LIN {X 0,Y 576.248,Z 853.833,A -85,B 0,C 180,E1 -7834.379,E2 -7834.379} C_VEL
LIN {X 0,Y 576.344,Z 849.843,A -85,B 0,C 180,E1 -7836.475,E2 -7836.475} C_VEL
LIN {X 0,Y 576.515,Z 844.122,A -85,B 0,C 180,E1 -7838.578,E2 -7838.578} C_VEL
LIN {X 0,Y 576.818,Z 836.801,A -85,B 0,C 180,E1 -7840.618,E2 -7840.618} C_VEL
LIN {X 0,Y 577.289,Z 827.415,A -85,B 0,C 180,E1 -7842.707,E2 -7842.707} C_VEL
LIN {X 0,Y 577.934,Z 816.921,A -85,B 0,C 180,E1 -7844.631,E2 -7844.631} C_VEL
LIN {X 0,Y 578.818,Z 804.354,A -85,B 0,C 180,E1 -7846.561,E2 -7846.561} C_VEL
LIN {X 0,Y 579.816,Z 790.982,A -85,B 0,C 180,E1 -7848.292,E2 -7848.292} C_VEL
LIN {X 0,Y 580.962,Z 776.343,A -85,B 0,C 180,E1 -7849.924,E2 -7849.924} C_VEL
LIN {X 0,Y 582.298,Z 759.809,A -85,B 0,C 180,E1 -7851.507,E2 -7851.507} C_VEL
LIN {X 0,Y 583.711,Z 742.222,A -85,B 0,C 180,E1 -7852.946,E2 -7852.946} C_VEL
LIN {X 0,Y 585.156,Z 723.193,A -85,B 0,C 180,E1 -7854.265,E2 -7854.265} C_VEL
LIN {X 0,Y 586.509,Z 703.816,A -85,B 0,C 180,E1 -7855.389,E2 -7855.389} C_VEL
LIN {X 0,Y 587.764,Z 683.712,A -85,B 0,C 180,E1 -7856.36,E2 -7856.36} C_VEL
LIN {X 0,Y 588.932,Z 661.915,A -85,B 0,C 180,E1 -7857.211,E2 -7857.211} C_VEL
LIN {X 0,Y 589.873,Z 640.331,A -85,B 0,C 180,E1 -7857.867,E2 -7857.867} C_VEL
LIN {X 0,Y 590.601,Z 617.84,A -85,B 0,C 180,E1 -7858.365,E2 -7858.365} C_VEL
LIN {X 0,Y 594.551,Z 503.519,A -85,B 0,C 180,E1 -7860.286,E2 -7860.286} C_VEL
LIN {X 0,Y 597.181,Z 414.489,A -85,B 0,C 180,E1 -7861.618,E2 -7861.618} C_VEL
LIN {X 0,Y 598.837,Z 339.586,A -85,B 0,C 180,E1 -7862.637,E2 -7862.637} C_VEL
LIN {X 0,Y 599.448,Z 336.228,A -85,B 0,C 180,E1 -7862.787,E2 -7862.787} C_VEL
LIN {X 0,Y 599.375,Z 306.855,A -85,B 0,C 180,E1 -7864.729,E2 -7864.729} C_VEL
LIN {X 0,Y 600.383,Z 268.326,A -85,B 0,C 180,E1 -7867.502,E2 -7867.502} C_VEL
LIN {X 0,Y 591.929,Z 246.123,A -85,B 0,C 180,E1 -7869.848,E2 -7869.848} C_VEL
LIN {X 0,Y 584.236,Z 228.435,A -85,B 0,C 180,E1 -7871.74,E2 -7871.74} C_VEL
LIN {X 0,Y 578.995,Z 217.335,A -85,B 0,C 180,E1 -7872.927,E2 -7872.927} C_VEL
LIN {X 0,Y 577.607,Z 214.744,A -85,B 0,C 180,E1 -7873.215,E2 -7873.215} C_VEL
LIN {X 0,Y 577.299,Z 213.311,A -85,B 0,C 180,E1 -7873.366,E2 -7873.366} C_VEL
LIN {X 0,Y 577.308,Z 213.309,A -85,B 0,C 180,E1 -7876.696,E2 -7876.696} C_VEL
LIN {X 0,Y 577.314,Z 213.308,A -85,B 0,C 180,E1 -7879.954,E2 -7879.954} C_VEL
LIN {X 0,Y 577.298,Z 213.305,A -85,B 0,C 180,E1 -7883.182,E2 -7883.182} C_VEL
LIN {X 0,Y 577.315,Z 213.304,A -85,B 0,C 180,E1 -7886.461,E2 -7886.461} C_VEL
LIN {X 0,Y 577.32,Z 213.314,A -85,B 0,C 180,E1 -7889.85,E2 -7889.85} C_VEL
LIN {X 0,Y 577.304,Z 213.311,A -85,B 0,C 180,E1 -7893.124,E2 -7893.124} C_VEL
LIN {X 0,Y 577.307,Z 213.291,A -85,B 0,C 180,E1 -7896.416,E2 -7896.416} C_VEL
LIN {X 0,Y 577.316,Z 213.314,A -85,B 0,C 180,E1 -7899.733,E2 -7899.733} C_VEL
LIN {X 0,Y 577.309,Z 213.299,A -85,B 0,C 180,E1 -7903.084,E2 -7903.084} C_VEL
LIN {X 0,Y 577.3,Z 213.303,A -85,B 0,C 180,E1 -7906.326,E2 -7906.326} C_VEL
LIN {X 0,Y 577.315,Z 213.307,A -85,B 0,C 180,E1 -7909.659,E2 -7909.659} C_VEL
LIN {X 0,Y 577.319,Z 213.3,A -85,B 0,C 180,E1 -7913.036,E2 -7913.036} C_VEL
LIN {X 0,Y 577.297,Z 213.318,A -85,B 0,C 180,E1 -7916.326,E2 -7916.326} C_VEL
LIN {X 0,Y 577.313,Z 213.295,A -85,B 0,C 180,E1 -7919.603,E2 -7919.603} C_VEL
LIN {X 0,Y 577.307,Z 213.312,A -85,B 0,C 180,E1 -7922.879,E2 -7922.879} C_VEL
LIN {X 0,Y 577.294,Z 213.294,A -85,B 0,C 180,E1 -7926.182,E2 -7926.182} C_VEL
LIN {X 0,Y 577.317,Z 213.31,A -85,B 0,C 180,E1 -7929.47,E2 -7929.47} C_VEL
LIN {X 0,Y 577.291,Z 213.316,A -85,B 0,C 180,E1 -7932.707,E2 -7932.707} C_VEL
LIN {X 0,Y 577.307,Z 213.316,A -85,B 0,C 180,E1 -7936.001,E2 -7936.001} C_VEL
LIN {X 0,Y 577.319,Z 213.312,A -85,B 0,C 180,E1 -7939.318,E2 -7939.318} C_VEL
LIN {X 0,Y 577.283,Z 213.322,A -85,B 0,C 180,E1 -7942.506,E2 -7942.506} C_VEL
LIN {X 0,Y 577.32,Z 213.321,A -85,B 0,C 180,E1 -7945.768,E2 -7945.768} C_VEL
LIN {X 0,Y 577.294,Z 213.316,A -85,B 0,C 180,E1 -7949.011,E2 -7949.011} C_VEL
LIN {X 0,Y 577.282,Z 213.322,A -85,B 0,C 180,E1 -7952.358,E2 -7952.358} C_VEL
LIN {X 0,Y 577.322,Z 213.313,A -85,B 0,C 180,E1 -7955.587,E2 -7955.587} C_VEL
LIN {X 0,Y 577.271,Z 213.322,A -85,B 0,C 180,E1 -7958.79,E2 -7958.79} C_VEL
LIN {X 0,Y 577.318,Z 213.515,A -85,B 0,C 180,E1 -7959.175,E2 -7959.175} C_VEL
LIN {X 0,Y 578.825,Z 217.068,A -85,B 0,C 180,E1 -7959.601,E2 -7959.601} C_VEL
LIN {X 0,Y 588.305,Z 235.653,A -85,B 0,C 180,E1 -7961.909,E2 -7961.909} C_VEL
LIN {X 0,Y 600.676,Z 260.638,A -85,B 0,C 180,E1 -7964.76,E2 -7964.76} C_VEL
LIN {X 0,Y 607.806,Z 275.644,A -85,B 0,C 180,E1 -7966.338,E2 -7966.338} C_VEL
LIN {X 0,Y 605.103,Z 308.798,A -85,B 0,C 180,E1 -7968.172,E2 -7968.172} C_VEL
LIN {X 0,Y 607.829,Z 331.377,A -85,B 0,C 180,E1 -7968.729,E2 -7968.729} C_VEL
LIN {X 0,Y 602.232,Z 577.23,A -85,B 0,C 180,E1 -7972.119,E2 -7972.119} C_VEL
LIN {X 0,Y 599.928,Z 692.589,A -85,B 0,C 180,E1 -7973.674,E2 -7973.674} C_VEL
LIN {X 0,Y 598.876,Z 717.126,A -85,B 0,C 180,E1 -7974.167,E2 -7974.167} C_VEL
LIN {X 0,Y 597.663,Z 738.821,A -85,B 0,C 180,E1 -7974.744,E2 -7974.744} C_VEL
LIN {X 0,Y 596.011,Z 763.246,A -85,B 0,C 180,E1 -7975.572,E2 -7975.572} C_VEL
LIN {X 0,Y 594.427,Z 783.289,A -85,B 0,C 180,E1 -7976.399,E2 -7976.399} C_VEL
LIN {X 0,Y 592.413,Z 806.84,A -85,B 0,C 180,E1 -7977.556,E2 -7977.556} C_VEL
LIN {X 0,Y 590.599,Z 826.305,A -85,B 0,C 180,E1 -7978.684,E2 -7978.684} C_VEL
LIN {X 0,Y 588.459,Z 848.134,A -85,B 0,C 180,E1 -7980.142,E2 -7980.142} C_VEL
LIN {X 0,Y 586.519,Z 867.008,A -85,B 0,C 180,E1 -7981.603,E2 -7981.603} C_VEL
LIN {X 0,Y 584.495,Z 887.006,A -85,B 0,C 180,E1 -7983.372,E2 -7983.372} C_VEL
LIN {X 0,Y 582.762,Z 903.916,A -85,B 0,C 180,E1 -7985.088,E2 -7985.088} C_VEL
LIN {X 0,Y 581.074,Z 921.418,A -85,B 0,C 180,E1 -7987.114,E2 -7987.114} C_VEL
LIN {X 0,Y 579.75,Z 935.465,A -85,B 0,C 180,E1 -7988.977,E2 -7988.977} C_VEL
LIN {X 0,Y 578.56,Z 949.769,A -85,B 0,C 180,E1 -7991.145,E2 -7991.145} C_VEL
LIN {X 0,Y 577.681,Z 961.419,A -85,B 0,C 180,E1 -7993.199,E2 -7993.199} C_VEL
LIN {X 0,Y 576.975,Z 972.466,A -85,B 0,C 180,E1 -7995.447,E2 -7995.447} C_VEL
LIN {X 0,Y 576.545,Z 980.188,A -85,B 0,C 180,E1 -7997.378,E2 -7997.378} C_VEL
LIN {X 0,Y 576.225,Z 987.119,A -85,B 0,C 180,E1 -7999.502,E2 -7999.502} C_VEL
LIN {X 0,Y 576.012,Z 993.449,A -85,B 0,C 180,E1 -8001.917,E2 -8001.917} C_VEL
LIN {X 0,Y 575.941,Z 997.697,A -85,B 0,C 180,E1 -8004.148,E2 -8004.148} C_VEL
LIN {X 0,Y 575.915,Z 1000.576,A -85,B 0,C 180,E1 -8006.317,E2 -8006.317} C_VEL
LIN {X 0,Y 575.907,Z 1002.235,A -85,B 0,C 180,E1 -8008.806,E2 -8008.806} C_VEL
LIN {X 0,Y 575.888,Z 1002.325,A -85,B 0,C 180,E1 -8010.796,E2 -8010.796} C_VEL
LIN {X 0,Y 575.886,Z 1001.289,A -85,B 0,C 180,E1 -8012.886,E2 -8012.886} C_VEL
LIN {X 0,Y 575.909,Z 998.45,A -85,B 0,C 180,E1 -8015.38,E2 -8015.38} C_VEL
LIN {X 0,Y 575.969,Z 994.688,A -85,B 0,C 180,E1 -8017.481,E2 -8017.481} C_VEL
LIN {X 0,Y 576.141,Z 989.457,A -85,B 0,C 180,E1 -8019.692,E2 -8019.692} C_VEL
LIN {X 0,Y 576.451,Z 981.951,A -85,B 0,C 180,E1 -8022.116,E2 -8022.116} C_VEL
LIN {X 0,Y 576.79,Z 975.298,A -85,B 0,C 180,E1 -8023.883,E2 -8023.883} C_VEL
LIN {X 0,Y 577.322,Z 966.57,A -85,B 0,C 180,E1 -8025.778,E2 -8025.778} C_VEL
LIN {X 0,Y 578.171,Z 954.305,A -85,B 0,C 180,E1 -8028.033,E2 -8028.033} C_VEL
LIN {X 0,Y 579.14,Z 941.931,A -85,B 0,C 180,E1 -8029.99,E2 -8029.99} C_VEL
LIN {X 0,Y 580.46,Z 926.019,A -85,B 0,C 180,E1 -8032.163,E2 -8032.163} C_VEL
LIN {X 0,Y 581.785,Z 911.136,A -85,B 0,C 180,E1 -8033.929,E2 -8033.929} C_VEL
LIN {X 0,Y 583.484,Z 892.287,A -85,B 0,C 180,E1 -8035.885,E2 -8035.885} C_VEL
LIN {X 0,Y 585.062,Z 875.137,A -85,B 0,C 180,E1 -8037.432,E2 -8037.432} C_VEL
LIN {X 0,Y 586.934,Z 854.247,A -85,B 0,C 180,E1 -8039.08,E2 -8039.08} C_VEL
LIN {X 0,Y 588.596,Z 834.717,A -85,B 0,C 180,E1 -8040.413,E2 -8040.413} C_VEL
LIN {X 0,Y 590.519,Z 811.335,A -85,B 0,C 180,E1 -8041.787,E2 -8041.787} C_VEL
LIN {X 0,Y 592.038,Z 790.551,A -85,B 0,C 180,E1 -8042.829,E2 -8042.829} C_VEL
LIN {X 0,Y 593.635,Z 766.597,A -85,B 0,C 180,E1 -8043.832,E2 -8043.832} C_VEL
LIN {X 0,Y 594.899,Z 744.933,A -85,B 0,C 180,E1 -8044.58,E2 -8044.58} C_VEL
LIN {X 0,Y 596.12,Z 719.728,A -85,B 0,C 180,E1 -8045.261,E2 -8045.261} C_VEL
LIN {X 0,Y 596.892,Z 698.83,A -85,B 0,C 180,E1 -8045.688,E2 -8045.688} C_VEL
LIN {X 0,Y 597.508,Z 665.557,A -85,B 0,C 180,E1 -8046.153,E2 -8046.153} C_VEL
LIN {X 0,Y 599.383,Z 523.368,A -85,B 0,C 180,E1 -8047.959,E2 -8047.959} C_VEL
LIN {X 0,Y 602.037,Z 398.059,A -85,B 0,C 180,E1 -8049.719,E2 -8049.719} C_VEL
LIN {X 0,Y 603.978,Z 328.15,A -85,B 0,C 180,E1 -8050.796,E2 -8050.796} C_VEL
LIN {X 0,Y 603.753,Z 324.587,A -85,B 0,C 180,E1 -8050.92,E2 -8050.92} C_VEL
LIN {X 0,Y 608.265,Z 300.685,A -85,B 0,C 180,E1 -8052.571,E2 -8052.571} C_VEL
LIN {X 0,Y 613.531,Z 280.646,A -85,B 0,C 180,E1 -8054.099,E2 -8054.099} C_VEL
LIN {X 0,Y 612.091,Z 275.219,A -85,B 0,C 180,E1 -8055.284,E2 -8055.284} C_VEL
LIN {X 0,Y 611.11,Z 271.585,A -85,B 0,C 180,E1 -8056.462,E2 -8056.462} C_VEL
LIN {X 0,Y 610.691,Z 269.324,A -85,B 0,C 180,E1 -8057.877,E2 -8057.877} C_VEL
LIN {X 0,Y 610.625,Z 269.272,A -85,B 0,C 180,E1 -8058.457,E2 -8058.457} C_VEL
LIN {X 0,Y 610.726,Z 271.372,A -85,B 0,C 180,E1 -8059.952,E2 -8059.952} C_VEL
LIN {X 0,Y 611.329,Z 275.332,A -85,B 0,C 180,E1 -8061.212,E2 -8061.212} C_VEL
LIN {X 0,Y 611.672,Z 278.803,A -85,B 0,C 180,E1 -8061.955,E2 -8061.955} C_VEL
LIN {X 0,Y 605.574,Z 300.252,A -85,B 0,C 180,E1 -8063.881,E2 -8063.881} C_VEL
LIN {X 0,Y 599.965,Z 327.92,A -85,B 0,C 180,E1 -8066.176,E2 -8066.176} C_VEL
LIN {X 0,Y 595.013,Z 362.924,A -85,B 0,C 180,E1 -8068.886,E2 -8068.886} C_VEL
LIN {X 0,Y 590.47,Z 407.602,A -85,B 0,C 180,E1 -8072.122,E2 -8072.122} C_VEL
LIN {X 0,Y 589.4,Z 422.994,A -85,B 0,C 180,E1 -8073.168,E2 -8073.168} C_VEL
LIN {X 0,Y 592.686,Z 455.008,A -85,B 0,C 180,E1 -8074.339,E2 -8074.339} C_VEL
LIN {X 0,Y 595.543,Z 491.146,A -85,B 0,C 180,E1 -8075.476,E2 -8075.476} C_VEL
LIN {X 0,Y 594.867,Z 505.645,A -85,B 0,C 180,E1 -8075.78,E2 -8075.78} C_VEL
LIN {X 0,Y 589.455,Z 607.464,A -85,B 0,C 180,E1 -8077.73,E2 -8077.73} C_VEL
LIN {X 0,Y 586.293,Z 687.572,A -85,B 0,C 180,E1 -8079.223,E2 -8079.223} C_VEL
LIN {X 0,Y 585.33,Z 709.905,A -85,B 0,C 180,E1 -8079.833,E2 -8079.833} C_VEL
LIN {X 0,Y 584.359,Z 731.272,A -85,B 0,C 180,E1 -8080.613,E2 -8080.613} C_VEL
LIN {X 0,Y 583.386,Z 750.706,A -85,B 0,C 180,E1 -8081.514,E2 -8081.514} C_VEL
LIN {X 0,Y 582.433,Z 769.003,A -85,B 0,C 180,E1 -8082.568,E2 -8082.568} C_VEL
LIN {X 0,Y 581.473,Z 786.178,A -85,B 0,C 180,E1 -8083.774,E2 -8083.774} C_VEL
LIN {X 0,Y 580.594,Z 801.262,A -85,B 0,C 180,E1 -8085.049,E2 -8085.049} C_VEL
LIN {X 0,Y 579.773,Z 814.876,A -85,B 0,C 180,E1 -8086.435,E2 -8086.435} C_VEL
LIN {X 0,Y 579.038,Z 827.147,A -85,B 0,C 180,E1 -8087.939,E2 -8087.939} C_VEL
LIN {X 0,Y 578.439,Z 837.273,A -85,B 0,C 180,E1 -8089.442,E2 -8089.442} C_VEL
LIN {X 0,Y 577.896,Z 846.496,A -85,B 0,C 180,E1 -8091.142,E2 -8091.142} C_VEL
LIN {X 0,Y 577.499,Z 853.707,A -85,B 0,C 180,E1 -8092.839,E2 -8092.839} C_VEL
LIN {X 0,Y 577.21,Z 859.389,A -85,B 0,C 180,E1 -8094.632,E2 -8094.632} C_VEL
LIN {X 0,Y 576.993,Z 863.232,A -85,B 0,C 180,E1 -8096.423,E2 -8096.423} C_VEL
LIN {X 0,Y 576.852,Z 865.342,A -85,B 0,C 180,E1 -8098.212,E2 -8098.212} C_VEL
LIN {X 0,Y 576.771,Z 865.736,A -85,B 0,C 180,E1 -8100.099,E2 -8100.099} C_VEL
LIN {X 0,Y 576.736,Z 864.293,A -85,B 0,C 180,E1 -8101.987,E2 -8101.987} C_VEL
LIN {X 0,Y 576.764,Z 861.014,A -85,B 0,C 180,E1 -8103.877,E2 -8103.877} C_VEL
LIN {X 0,Y 576.874,Z 856.161,A -85,B 0,C 180,E1 -8105.67,E2 -8105.67} C_VEL
LIN {X 0,Y 577.061,Z 849.471,A -85,B 0,C 180,E1 -8107.467,E2 -8107.467} C_VEL
LIN {X 0,Y 577.367,Z 841.126,A -85,B 0,C 180,E1 -8109.201,E2 -8109.201} C_VEL
LIN {X 0,Y 577.814,Z 831.101,A -85,B 0,C 180,E1 -8110.872,E2 -8110.872} C_VEL
LIN {X 0,Y 578.397,Z 819.329,A -85,B 0,C 180,E1 -8112.48,E2 -8112.48} C_VEL
LIN {X 0,Y 579.11,Z 805.98,A -85,B 0,C 180,E1 -8113.988,E2 -8113.988} C_VEL
LIN {X 0,Y 579.937,Z 790.987,A -85,B 0,C 180,E1 -8115.398,E2 -8115.398} C_VEL
LIN {X 0,Y 580.827,Z 774.875,A -85,B 0,C 180,E1 -8116.656,E2 -8116.656} C_VEL
LIN {X 0,Y 581.733,Z 757.436,A -85,B 0,C 180,E1 -8117.782,E2 -8117.782} C_VEL
LIN {X 0,Y 582.635,Z 739.626,A -85,B 0,C 180,E1 -8118.719,E2 -8118.719} C_VEL
LIN {X 0,Y 583.514,Z 720.275,A -85,B 0,C 180,E1 -8119.531,E2 -8119.531} C_VEL
LIN {X 0,Y 584.279,Z 700.12,A -85,B 0,C 180,E1 -8120.172,E2 -8120.172} C_VEL
LIN {X 0,Y 584.919,Z 679.428,A -85,B 0,C 180,E1 -8120.63,E2 -8120.63} C_VEL
LIN {X 0,Y 588.981,Z 489.215,A -85,B 0,C 180,E1 -8123.466,E2 -8123.466} C_VEL
LIN {X 0,Y 585.221,Z 455.543,A -85,B 0,C 180,E1 -8124.209,E2 -8124.209} C_VEL
LIN {X 0,Y 587.587,Z 405.605,A -85,B 0,C 180,E1 -8127.406,E2 -8127.406} C_VEL
LIN {X 0,Y 590.441,Z 352.546,A -85,B 0,C 180,E1 -8130.842,E2 -8130.842} C_VEL
LIN {X 0,Y 593.46,Z 300.77,A -85,B 0,C 180,E1 -8134.246,E2 -8134.246} C_VEL
LIN {X 0,Y 595.914,Z 261.134,A -85,B 0,C 180,E1 -8136.892,E2 -8136.892} C_VEL
LIN {X 0,Y 591.877,Z 250.242,A -85,B 0,C 180,E1 -8137.944,E2 -8137.944} C_VEL
LIN {X 0,Y 589.101,Z 245.546,A -85,B 0,C 180,E1 -8138.478,E2 -8138.478} C_VEL
LIN {X 0,Y 577.793,Z 233.961,A -85,B 0,C 180,E1 -8140.148,E2 -8140.148} C_VEL
LIN {X 0,Y 576.198,Z 231.311,A -85,B 0,C 180,E1 -8140.468,E2 -8140.468} C_VEL
LIN {X 0,Y 569.344,Z 214.421,A -85,B 0,C 180,E1 -8142.302,E2 -8142.302} C_VEL
LIN {X 0,Y 569.381,Z 214.302,A -85,B 0,C 180,E1 -8145.518,E2 -8145.518} C_VEL
LIN {X 0,Y 569.39,Z 214.435,A -85,B 0,C 180,E1 -8146.119,E2 -8146.119} C_VEL
LIN {X 0,Y 570.341,Z 217.235,A -85,B 0,C 180,E1 -8146.39,E2 -8146.39} C_VEL
LIN {X 0,Y 571.71,Z 219.791,A -85,B 0,C 180,E1 -8146.683,E2 -8146.683} C_VEL
LIN {X 0,Y 578.876,Z 234.711,A -85,B 0,C 180,E1 -8148.317,E2 -8148.317} C_VEL
LIN {X 0,Y 586.838,Z 253.704,A -85,B 0,C 180,E1 -8150.367,E2 -8150.367} C_VEL
LIN {X 0,Y 593.746,Z 272.147,A -85,B 0,C 180,E1 -8152.326,E2 -8152.326} C_VEL
LIN {X 0,Y 592.76,Z 314.667,A -85,B 0,C 180,E1 -8155.357,E2 -8155.357} C_VEL
LIN {X 0,Y 592.824,Z 338.961,A -85,B 0,C 180,E1 -8156.932,E2 -8156.932} C_VEL
LIN {X 0,Y 591.933,Z 343.747,A -85,B 0,C 180,E1 -8157.101,E2 -8157.101} C_VEL
LIN {X 0,Y 589.728,Z 439.794,A -85,B 0,C 180,E1 -8158.419,E2 -8158.419} C_VEL
LIN {X 0,Y 586.74,Z 530.066,A -85,B 0,C 180,E1 -8159.837,E2 -8159.837} C_VEL
LIN {X 0,Y 583.259,Z 625.148,A -85,B 0,C 180,E1 -8161.508,E2 -8161.508} C_VEL
LIN {X 0,Y 582.489,Z 647.168,A -85,B 0,C 180,E1 -8162.048,E2 -8162.048} C_VEL
LIN {X 0,Y 581.453,Z 668.771,A -85,B 0,C 180,E1 -8162.755,E2 -8162.755} C_VEL
LIN {X 0,Y 580.207,Z 690.159,A -85,B 0,C 180,E1 -8163.655,E2 -8163.655} C_VEL
LIN {X 0,Y 578.823,Z 710.131,A -85,B 0,C 180,E1 -8164.688,E2 -8164.688} C_VEL
LIN {X 0,Y 577.378,Z 729.317,A -85,B 0,C 180,E1 -8165.877,E2 -8165.877} C_VEL
LIN {X 0,Y 575.82,Z 748.322,A -85,B 0,C 180,E1 -8167.272,E2 -8167.272} C_VEL
LIN {X 0,Y 574.417,Z 765.121,A -85,B 0,C 180,E1 -8168.719,E2 -8168.719} C_VEL
LIN {X 0,Y 573.057,Z 781.033,A -85,B 0,C 180,E1 -8170.321,E2 -8170.321} C_VEL
LIN {X 0,Y 571.809,Z 795.88,A -85,B 0,C 180,E1 -8172.076,E2 -8172.076} C_VEL
LIN {X 0,Y 570.757,Z 809.256,A -85,B 0,C 180,E1 -8173.931,E2 -8173.931} C_VEL
LIN {X 0,Y 569.863,Z 821.736,A -85,B 0,C 180,E1 -8175.987,E2 -8175.987} C_VEL
LIN {X 0,Y 569.248,Z 831.607,A -85,B 0,C 180,E1 -8177.935,E2 -8177.935} C_VEL
LIN {X 0,Y 568.806,Z 840.094,A -85,B 0,C 180,E1 -8179.978,E2 -8179.978} C_VEL
LIN {X 0,Y 568.521,Z 846.753,A -85,B 0,C 180,E1 -8182.013,E2 -8182.013} C_VEL
LIN {X 0,Y 568.361,Z 852.257,A -85,B 0,C 180,E1 -8184.245,E2 -8184.245} C_VEL
LIN {X 0,Y 568.297,Z 855.835,A -85,B 0,C 180,E1 -8186.368,E2 -8186.368} C_VEL
LIN {X 0,Y 568.26,Z 857.744,A -85,B 0,C 180,E1 -8188.488,E2 -8188.488} C_VEL
LIN {X 0,Y 568.247,Z 858.093,A -85,B 0,C 180,E1 -8190.605,E2 -8190.605} C_VEL
LIN {X 0,Y 568.274,Z 856.938,A -85,B 0,C 180,E1 -8192.723,E2 -8192.723} C_VEL
LIN {X 0,Y 568.33,Z 854.144,A -85,B 0,C 180,E1 -8194.844,E2 -8194.844} C_VEL
LIN {X 0,Y 568.421,Z 849.713,A -85,B 0,C 180,E1 -8196.971,E2 -8196.971} C_VEL
LIN {X 0,Y 568.641,Z 843.588,A -85,B 0,C 180,E1 -8199.106,E2 -8199.106} C_VEL
LIN {X 0,Y 569.027,Z 836.048,A -85,B 0,C 180,E1 -8201.145,E2 -8201.145} C_VEL
LIN {X 0,Y 569.547,Z 826.578,A -85,B 0,C 180,E1 -8203.193,E2 -8203.193} C_VEL
LIN {X 0,Y 570.279,Z 815.707,A -85,B 0,C 180,E1 -8205.144,E2 -8205.144} C_VEL
LIN {X 0,Y 571.203,Z 803.495,A -85,B 0,C 180,E1 -8206.998,E2 -8206.998} C_VEL
LIN {X 0,Y 572.319,Z 789.976,A -85,B 0,C 180,E1 -8208.751,E2 -8208.751} C_VEL
LIN {X 0,Y 573.661,Z 774.003,A -85,B 0,C 180,E1 -8210.508,E2 -8210.508} C_VEL
LIN {X 0,Y 575.071,Z 757.356,A -85,B 0,C 180,E1 -8212.067,E2 -8212.067} C_VEL
LIN {X 0,Y 576.568,Z 739.348,A -85,B 0,C 180,E1 -8213.507,E2 -8213.507} C_VEL
LIN {X 0,Y 578.148,Z 719.445,A -85,B 0,C 180,E1 -8214.851,E2 -8214.851} C_VEL
LIN {X 0,Y 579.515,Z 700.296,A -85,B 0,C 180,E1 -8215.937,E2 -8215.937} C_VEL
LIN {X 0,Y 580.878,Z 679.328,A -85,B 0,C 180,E1 -8216.918,E2 -8216.918} C_VEL
LIN {X 0,Y 581.989,Z 658.553,A -85,B 0,C 180,E1 -8217.693,E2 -8217.693} C_VEL
LIN {X 0,Y 582.878,Z 636.878,A -85,B 0,C 180,E1 -8218.318,E2 -8218.318} C_VEL
LIN {X 0,Y 583.753,Z 609.709,A -85,B 0,C 180,E1 -8218.876,E2 -8218.876} C_VEL
LIN {X 0,Y 587.697,Z 503.594,A -85,B 0,C 180,E1 -8220.688,E2 -8220.688} C_VEL
LIN {X 0,Y 590.36,Z 417.842,A -85,B 0,C 180,E1 -8221.989,E2 -8221.989} C_VEL
LIN {X 0,Y 591.983,Z 342.833,A -85,B 0,C 180,E1 -8223.005,E2 -8223.005} C_VEL
LIN {X 0,Y 592.926,Z 337.654,A -85,B 0,C 180,E1 -8223.235,E2 -8223.235} C_VEL
LIN {X 0,Y 592.875,Z 307.651,A -85,B 0,C 180,E1 -8225.225,E2 -8225.225} C_VEL
LIN {X 0,Y 593.748,Z 271.834,A -85,B 0,C 180,E1 -8227.806,E2 -8227.806} C_VEL
LIN {X 0,Y 585.364,Z 249.888,A -85,B 0,C 180,E1 -8230.146,E2 -8230.146} C_VEL
LIN {X 0,Y 578.158,Z 233.181,A -85,B 0,C 180,E1 -8231.956,E2 -8231.956} C_VEL
LIN {X 0,Y 571.21,Z 218.485,A -85,B 0,C 180,E1 -8233.556,E2 -8233.556} C_VEL
LIN {X 0,Y 569.605,Z 215.436,A -85,B 0,C 180,E1 -8233.899,E2 -8233.899} C_VEL
LIN {X 0,Y 569.377,Z 214.299,A -85,B 0,C 180,E1 -8234.026,E2 -8234.026} C_VEL
LIN {X 0,Y 569.36,Z 214.306,A -85,B 0,C 180,E1 -8237.322,E2 -8237.322} C_VEL
LIN {X 0,Y 569.378,Z 214.305,A -85,B 0,C 180,E1 -8240.657,E2 -8240.657} C_VEL
LIN {X 0,Y 569.374,Z 214.297,A -85,B 0,C 180,E1 -8243.963,E2 -8243.963} C_VEL
LIN {X 0,Y 569.361,Z 214.289,A -85,B 0,C 180,E1 -8247.267,E2 -8247.267} C_VEL
LIN {X 0,Y 569.38,Z 214.295,A -85,B 0,C 180,E1 -8250.578,E2 -8250.578} C_VEL
LIN {X 0,Y 569.374,Z 214.308,A -85,B 0,C 180,E1 -8253.958,E2 -8253.958} C_VEL
LIN {X 0,Y 569.365,Z 214.284,A -85,B 0,C 180,E1 -8257.272,E2 -8257.272} C_VEL
LIN {X 0,Y 569.371,Z 214.293,A -85,B 0,C 180,E1 -8260.569,E2 -8260.569} C_VEL
LIN {X 0,Y 569.372,Z 214.303,A -85,B 0,C 180,E1 -8263.995,E2 -8263.995} C_VEL
LIN {X 0,Y 569.369,Z 214.281,A -85,B 0,C 180,E1 -8267.216,E2 -8267.216} C_VEL
LIN {X 0,Y 569.363,Z 214.305,A -85,B 0,C 180,E1 -8270.498,E2 -8270.498} C_VEL
LIN {X 0,Y 569.374,Z 214.277,A -85,B 0,C 180,E1 -8273.85,E2 -8273.85} C_VEL
LIN {X 0,Y 569.376,Z 214.304,A -85,B 0,C 180,E1 -8277.182,E2 -8277.182} C_VEL
LIN {X 0,Y 569.352,Z 214.275,A -85,B 0,C 180,E1 -8280.402,E2 -8280.402} C_VEL
LIN {X 0,Y 569.376,Z 214.308,A -85,B 0,C 180,E1 -8283.725,E2 -8283.725} C_VEL
LIN {X 0,Y 569.38,Z 214.272,A -85,B 0,C 180,E1 -8287.061,E2 -8287.061} C_VEL
LIN {X 0,Y 569.35,Z 214.308,A -85,B 0,C 180,E1 -8290.422,E2 -8290.422} C_VEL
LIN {X 0,Y 569.382,Z 214.308,A -85,B 0,C 180,E1 -8293.714,E2 -8293.714} C_VEL
LIN {X 0,Y 569.361,Z 214.306,A -85,B 0,C 180,E1 -8296.949,E2 -8296.949} C_VEL
LIN {X 0,Y 569.348,Z 214.308,A -85,B 0,C 180,E1 -8300.349,E2 -8300.349} C_VEL
LIN {X 0,Y 569.383,Z 214.305,A -85,B 0,C 180,E1 -8303.603,E2 -8303.603} C_VEL
LIN {X 0,Y 569.346,Z 214.301,A -85,B 0,C 180,E1 -8306.855,E2 -8306.855} C_VEL
LIN {X 0,Y 569.353,Z 214.312,A -85,B 0,C 180,E1 -8310.226,E2 -8310.226} C_VEL
LIN {X 0,Y 569.381,Z 214.303,A -85,B 0,C 180,E1 -8313.473,E2 -8313.473} C_VEL
LIN {X 0,Y 569.334,Z 214.309,A -85,B 0,C 180,E1 -8316.664,E2 -8316.664} C_VEL
LIN {X 0,Y 569.358,Z 214.444,A -85,B 0,C 180,E1 -8318.406,E2 -8318.406} C_VEL
LIN {X 0,Y 570.387,Z 217.397,A -85,B 0,C 180,E1 -8318.743,E2 -8318.743} C_VEL
LIN {X 0,Y 571.764,Z 219.658,A -85,B 0,C 180,E1 -8319.063,E2 -8319.063} C_VEL
LIN {X 0,Y 581.042,Z 238.068,A -85,B 0,C 180,E1 -8321.384,E2 -8321.384} C_VEL
LIN {X 0,Y 592.456,Z 260.848,A -85,B 0,C 180,E1 -8324.054,E2 -8324.054} C_VEL
LIN {X 0,Y 601.171,Z 279.402,A -85,B 0,C 180,E1 -8326.036,E2 -8326.036} C_VEL
LIN {X 0,Y 598.614,Z 309.394,A -85,B 0,C 180,E1 -8327.71,E2 -8327.71} C_VEL
LIN {X 0,Y 601.382,Z 332.717,A -85,B 0,C 180,E1 -8328.291,E2 -8328.291} C_VEL
LIN {X 0,Y 595.541,Z 572.332,A -85,B 0,C 180,E1 -8331.646,E2 -8331.646} C_VEL
LIN {X 0,Y 592.986,Z 692.835,A -85,B 0,C 180,E1 -8333.293,E2 -8333.293} C_VEL
LIN {X 0,Y 591.882,Z 717.267,A -85,B 0,C 180,E1 -8333.79,E2 -8333.79} C_VEL
LIN {X 0,Y 590.638,Z 738.58,A -85,B 0,C 180,E1 -8334.363,E2 -8334.363} C_VEL
LIN {X 0,Y 588.881,Z 763.35,A -85,B 0,C 180,E1 -8335.214,E2 -8335.214} C_VEL
LIN {X 0,Y 587.231,Z 783.315,A -85,B 0,C 180,E1 -8336.048,E2 -8336.048} C_VEL
LIN {X 0,Y 585.054,Z 807.455,A -85,B 0,C 180,E1 -8337.254,E2 -8337.254} C_VEL
LIN {X 0,Y 583.145,Z 827.122,A -85,B 0,C 180,E1 -8338.411,E2 -8338.411} C_VEL
LIN {X 0,Y 580.833,Z 849.426,A -85,B 0,C 180,E1 -8339.937,E2 -8339.937} C_VEL
LIN {X 0,Y 578.942,Z 867.051,A -85,B 0,C 180,E1 -8341.327,E2 -8341.327} C_VEL
LIN {X 0,Y 576.775,Z 887.323,A -85,B 0,C 180,E1 -8343.154,E2 -8343.154} C_VEL
LIN {X 0,Y 575.028,Z 903.654,A -85,B 0,C 180,E1 -8344.84,E2 -8344.84} C_VEL
LIN {X 0,Y 573.254,Z 921.098,A -85,B 0,C 180,E1 -8346.893,E2 -8346.893} C_VEL
LIN {X 0,Y 571.882,Z 935.11,A -85,B 0,C 180,E1 -8348.782,E2 -8348.782} C_VEL
LIN {X 0,Y 570.586,Z 949.964,A -85,B 0,C 180,E1 -8351.083,E2 -8351.083} C_VEL
LIN {X 0,Y 569.728,Z 960.976,A -85,B 0,C 180,E1 -8353.062,E2 -8353.062} C_VEL
LIN {X 0,Y 568.973,Z 972.391,A -85,B 0,C 180,E1 -8355.445,E2 -8355.445} C_VEL
LIN {X 0,Y 568.499,Z 980.992,A -85,B 0,C 180,E1 -8357.609,E2 -8357.609} C_VEL
LIN {X 0,Y 568.169,Z 988.802,A -85,B 0,C 180,E1 -8359.967,E2 -8359.967} C_VEL
LIN {X 0,Y 567.986,Z 994.275,A -85,B 0,C 180,E1 -8362.21,E2 -8362.21} C_VEL
LIN {X 0,Y 567.934,Z 997.972,A -85,B 0,C 180,E1 -8364.241,E2 -8364.241} C_VEL
LIN {X 0,Y 567.903,Z 1001.015,A -85,B 0,C 180,E1 -8366.669,E2 -8366.669} C_VEL
LIN {X 0,Y 567.898,Z 1002.28,A -85,B 0,C 180,E1 -8368.991,E2 -8368.991} C_VEL
LIN {X 0,Y 567.898,Z 1002.28,A -85,B 0,C 180,E1 -8371.009,E2 -8371.009} C_VEL
LIN {X 0,Y 567.906,Z 1000.915,A -85,B 0,C 180,E1 -8373.432,E2 -8373.432} C_VEL
LIN {X 0,Y 567.934,Z 997.971,A -85,B 0,C 180,E1 -8375.76,E2 -8375.76} C_VEL
LIN {X 0,Y 567.993,Z 994.069,A -85,B 0,C 180,E1 -8377.892,E2 -8377.892} C_VEL
LIN {X 0,Y 568.191,Z 988.158,A -85,B 0,C 180,E1 -8380.238,E2 -8380.238} C_VEL
LIN {X 0,Y 568.5,Z 980.91,A -85,B 0,C 180,E1 -8382.391,E2 -8382.391} C_VEL
LIN {X 0,Y 568.978,Z 972.186,A -85,B 0,C 180,E1 -8384.555,E2 -8384.555} C_VEL
LIN {X 0,Y 569.688,Z 961.092,A -85,B 0,C 180,E1 -8386.834,E2 -8386.834} C_VEL
LIN {X 0,Y 570.533,Z 949.674,A -85,B 0,C 180,E1 -8388.847,E2 -8388.847} C_VEL
LIN {X 0,Y 571.694,Z 935.436,A -85,B 0,C 180,E1 -8391.011,E2 -8391.011} C_VEL
LIN {X 0,Y 572.997,Z 921.077,A -85,B 0,C 180,E1 -8392.901,E2 -8392.901} C_VEL
LIN {X 0,Y 574.602,Z 903.659,A -85,B 0,C 180,E1 -8394.905,E2 -8394.905} C_VEL
LIN {X 0,Y 576.157,Z 887.303,A -85,B 0,C 180,E1 -8396.544,E2 -8396.544} C_VEL
LIN {X 0,Y 577.957,Z 868.083,A -85,B 0,C 180,E1 -8398.24,E2 -8398.24} C_VEL
LIN {X 0,Y 579.754,Z 848.643,A -85,B 0,C 180,E1 -8399.726,E2 -8399.726} C_VEL
LIN {X 0,Y 581.774,Z 826.231,A -85,B 0,C 180,E1 -8401.211,E2 -8401.211} C_VEL
LIN {X 0,Y 583.371,Z 806.617,A -85,B 0,C 180,E1 -8402.328,E2 -8402.328} C_VEL
LIN {X 0,Y 585.213,Z 782.574,A -85,B 0,C 180,E1 -8403.496,E2 -8403.496} C_VEL
LIN {X 0,Y 586.653,Z 761.498,A -85,B 0,C 180,E1 -8404.344,E2 -8404.344} C_VEL
LIN {X 0,Y 588.123,Z 736.576,A -85,B 0,C 180,E1 -8405.164,E2 -8405.164} C_VEL
LIN {X 0,Y 589.14,Z 714.548,A -85,B 0,C 180,E1 -8405.726,E2 -8405.726} C_VEL
LIN {X 0,Y 590.03,Z 688.498,A -85,B 0,C 180,E1 -8406.211,E2 -8406.211} C_VEL
LIN {X 0,Y 592.517,Z 526.417,A -85,B 0,C 180,E1 -8408.323,E2 -8408.323} C_VEL
LIN {X 0,Y 595.353,Z 407.844,A -85,B 0,C 180,E1 -8410.036,E2 -8410.036} C_VEL
LIN {X 0,Y 597.915,Z 329.601,A -85,B 0,C 180,E1 -8411.28,E2 -8411.28} C_VEL
LIN {X 0,Y 597.763,Z 327.352,A -85,B 0,C 180,E1 -8411.355,E2 -8411.355} C_VEL
LIN {X 0,Y 602.798,Z 303.687,A -85,B 0,C 180,E1 -8413.045,E2 -8413.045} C_VEL
LIN {X 0,Y 608.154,Z 285.464,A -85,B 0,C 180,E1 -8414.475,E2 -8414.475} C_VEL
LIN {X 0,Y 607.008,Z 280.361,A -85,B 0,C 180,E1 -8415.698,E2 -8415.698} C_VEL
LIN {X 0,Y 606.272,Z 277.736,A -85,B 0,C 180,E1 -8416.679,E2 -8416.679} C_VEL
LIN {X 0,Y 606.126,Z 275.632,A -85,B 0,C 180,E1 -8418.214,E2 -8418.214} C_VEL
LIN {X 0,Y 605.897,Z 277.499,A -85,B 0,C 180,E1 -8419.691,E2 -8419.691} C_VEL
LIN {X 0,Y 606.251,Z 280.584,A -85,B 0,C 180,E1 -8420.825,E2 -8420.825} C_VEL
LIN {X 0,Y 606.491,Z 283.655,A -85,B 0,C 180,E1 -8421.571,E2 -8421.571} C_VEL
LIN {X 0,Y 599.82,Z 304.959,A -85,B 0,C 180,E1 -8423.538,E2 -8423.538} C_VEL
LIN {X 0,Y 593.809,Z 331.937,A -85,B 0,C 180,E1 -8425.836,E2 -8425.836} C_VEL
LIN {X 0,Y 588.656,Z 364.932,A -85,B 0,C 180,E1 -8428.455,E2 -8428.455} C_VEL
LIN {X 0,Y 583.914,Z 406.935,A -85,B 0,C 180,E1 -8431.572,E2 -8431.572} C_VEL
LIN {X 0,Y 582.884,Z 419.506,A -85,B 0,C 180,E1 -8432.447,E2 -8432.447} C_VEL
LIN {X 0,Y 585.632,Z 446.596,A -85,B 0,C 180,E1 -8433.505,E2 -8433.505} C_VEL
LIN {X 0,Y 588.405,Z 481.333,A -85,B 0,C 180,E1 -8434.69,E2 -8434.69} C_VEL
LIN {X 0,Y 589.088,Z 495.815,A -85,B 0,C 180,E1 -8435.116,E2 -8435.116} C_VEL
LIN {X 0,Y 583.019,Z 598.12,A -85,B 0,C 180,E1 -8437.152,E2 -8437.152} C_VEL
LIN {X 0,Y 579.118,Z 687.482,A -85,B 0,C 180,E1 -8438.87,E2 -8438.87} C_VEL
LIN {X 0,Y 578.059,Z 710.48,A -85,B 0,C 180,E1 -8439.509,E2 -8439.509} C_VEL
LIN {X 0,Y 577.073,Z 730.613,A -85,B 0,C 180,E1 -8440.252,E2 -8440.252} C_VEL
LIN {X 0,Y 576.021,Z 750.164,A -85,B 0,C 180,E1 -8441.163,E2 -8441.163} C_VEL
LIN {X 0,Y 575.015,Z 768.532,A -85,B 0,C 180,E1 -8442.215,E2 -8442.215} C_VEL
LIN {X 0,Y 574.02,Z 785.524,A -85,B 0,C 180,E1 -8443.401,E2 -8443.401} C_VEL
LIN {X 0,Y 573.042,Z 801.208,A -85,B 0,C 180,E1 -8444.723,E2 -8444.723} C_VEL
LIN {X 0,Y 572.151,Z 815.237,A -85,B 0,C 180,E1 -8446.148,E2 -8446.148} C_VEL
LIN {X 0,Y 571.352,Z 827.64,A -85,B 0,C 180,E1 -8447.672,E2 -8447.672} C_VEL
LIN {X 0,Y 570.654,Z 838.462,A -85,B 0,C 180,E1 -8449.296,E2 -8449.296} C_VEL
LIN {X 0,Y 570.107,Z 847.239,A -85,B 0,C 180,E1 -8450.918,E2 -8450.918} C_VEL
LIN {X 0,Y 569.668,Z 854.55,A -85,B 0,C 180,E1 -8452.638,E2 -8452.638} C_VEL
LIN {X 0,Y 569.345,Z 860.304,A -85,B 0,C 180,E1 -8454.457,E2 -8454.457} C_VEL
LIN {X 0,Y 569.089,Z 864.343,A -85,B 0,C 180,E1 -8456.357,E2 -8456.357} C_VEL
LIN {X 0,Y 568.932,Z 866.445,A -85,B 0,C 180,E1 -8458.187,E2 -8458.187} C_VEL
LIN {X 0,Y 568.841,Z 866.79,A -85,B 0,C 180,E1 -8460.101,E2 -8460.101} C_VEL
LIN {X 0,Y 568.802,Z 865.285,A -85,B 0,C 180,E1 -8462.015,E2 -8462.015} C_VEL
LIN {X 0,Y 568.828,Z 862.171,A -85,B 0,C 180,E1 -8463.83,E2 -8463.83} C_VEL
LIN {X 0,Y 568.939,Z 857.335,A -85,B 0,C 180,E1 -8465.648,E2 -8465.648} C_VEL
LIN {X 0,Y 569.132,Z 850.663,A -85,B 0,C 180,E1 -8467.47,E2 -8467.47} C_VEL
LIN {X 0,Y 569.443,Z 842.522,A -85,B 0,C 180,E1 -8469.195,E2 -8469.195} C_VEL
LIN {X 0,Y 569.912,Z 832.342,A -85,B 0,C 180,E1 -8470.923,E2 -8470.923} C_VEL
LIN {X 0,Y 570.518,Z 820.608,A -85,B 0,C 180,E1 -8472.552,E2 -8472.552} C_VEL
LIN {X 0,Y 571.257,Z 807.31,A -85,B 0,C 180,E1 -8474.081,E2 -8474.081} C_VEL
LIN {X 0,Y 572.113,Z 792.39,A -85,B 0,C 180,E1 -8475.51,E2 -8475.51} C_VEL
LIN {X 0,Y 573.037,Z 776.385,A -85,B 0,C 180,E1 -8476.785,E2 -8476.785} C_VEL
LIN {X 0,Y 573.957,Z 759.406,A -85,B 0,C 180,E1 -8477.908,E2 -8477.908} C_VEL
LIN {X 0,Y 574.926,Z 741.101,A -85,B 0,C 180,E1 -8478.896,E2 -8478.896} C_VEL
LIN {X 0,Y 575.801,Z 722.815,A -85,B 0,C 180,E1 -8479.687,E2 -8479.687} C_VEL
LIN {X 0,Y 576.605,Z 703.153,A -85,B 0,C 180,E1 -8480.346,E2 -8480.346} C_VEL
LIN {X 0,Y 577.304,Z 682.763,A -85,B 0,C 180,E1 -8480.837,E2 -8480.837} C_VEL
LIN {X 0,Y 581.678,Z 489.866,A -85,B 0,C 180,E1 -8483.789,E2 -8483.789} C_VEL
LIN {X 0,Y 577.785,Z 454.855,A -85,B 0,C 180,E1 -8484.568,E2 -8484.568} C_VEL
LIN {X 0,Y 580.371,Z 403.516,A -85,B 0,C 180,E1 -8487.893,E2 -8487.893} C_VEL
LIN {X 0,Y 583.308,Z 351.623,A -85,B 0,C 180,E1 -8491.292,E2 -8491.292} C_VEL
LIN {X 0,Y 586.526,Z 299.648,A -85,B 0,C 180,E1 -8494.745,E2 -8494.745} C_VEL
LIN {X 0,Y 588.85,Z 264.23,A -85,B 0,C 180,E1 -8497.133,E2 -8497.133} C_VEL
LIN {X 0,Y 580.082,Z 241.04,A -85,B 0,C 180,E1 -8499.446,E2 -8499.446} C_VEL
LIN {X 0,Y 576.198,Z 231.311,A -85,B 0,C 180,E1 -8500.468,E2 -8500.468} C_VEL
LIN {X 0,Y 573.888,Z 228.587,A -85,B 0,C 180,E1 -8500.85,E2 -8500.85} C_VEL
LIN {X 0,Y 565.359,Z 223.504,A -85,B 0,C 180,E1 -8501.905,E2 -8501.905} C_VEL
LIN {X 0,Y 563.532,Z 221.076,A -85,B 0,C 180,E1 -8502.24,E2 -8502.24} C_VEL
LIN {X 0,Y 561.425,Z 215.295,A -85,B 0,C 180,E1 -8502.905,E2 -8502.905} C_VEL
LIN {X 0,Y 561.47,Z 215.494,A -85,B 0,C 180,E1 -8505.44,E2 -8505.44} C_VEL
LIN {X 0,Y 562.583,Z 218.532,A -85,B 0,C 180,E1 -8505.747,E2 -8505.747} C_VEL
LIN {X 0,Y 563.947,Z 221.073,A -85,B 0,C 180,E1 -8506.042,E2 -8506.042} C_VEL
LIN {X 0,Y 571.17,Z 235.872,A -85,B 0,C 180,E1 -8507.7,E2 -8507.7} C_VEL
LIN {X 0,Y 578.648,Z 253.223,A -85,B 0,C 180,E1 -8509.61,E2 -8509.61} C_VEL
LIN {X 0,Y 587.03,Z 275.288,A -85,B 0,C 180,E1 -8511.979,E2 -8511.979} C_VEL
LIN {X 0,Y 586.494,Z 302.823,A -85,B 0,C 180,E1 -8513.972,E2 -8513.972} C_VEL
LIN {X 0,Y 586.337,Z 334.407,A -85,B 0,C 180,E1 -8516.107,E2 -8516.107} C_VEL
LIN {X 0,Y 586.342,Z 340.65,A -85,B 0,C 180,E1 -8516.492,E2 -8516.492} C_VEL
LIN {X 0,Y 585.23,Z 346.433,A -85,B 0,C 180,E1 -8516.701,E2 -8516.701} C_VEL
LIN {X 0,Y 582.959,Z 441.18,A -85,B 0,C 180,E1 -8518.015,E2 -8518.015} C_VEL
LIN {X 0,Y 579.921,Z 528.99,A -85,B 0,C 180,E1 -8519.413,E2 -8519.413} C_VEL
LIN {X 0,Y 576.179,Z 625.533,A -85,B 0,C 180,E1 -8521.141,E2 -8521.141} C_VEL
LIN {X 0,Y 575.409,Z 647.412,A -85,B 0,C 180,E1 -8521.677,E2 -8521.677} C_VEL
LIN {X 0,Y 574.297,Z 669.63,A -85,B 0,C 180,E1 -8522.411,E2 -8522.411} C_VEL
LIN {X 0,Y 573.012,Z 690.725,A -85,B 0,C 180,E1 -8523.308,E2 -8523.308} C_VEL
LIN {X 0,Y 571.579,Z 710.623,A -85,B 0,C 180,E1 -8524.344,E2 -8524.344} C_VEL
LIN {X 0,Y 569.998,Z 730.666,A -85,B 0,C 180,E1 -8525.599,E2 -8525.599} C_VEL
LIN {X 0,Y 568.423,Z 748.96,A -85,B 0,C 180,E1 -8526.959,E2 -8526.959} C_VEL
LIN {X 0,Y 566.939,Z 765.82,A -85,B 0,C 180,E1 -8528.425,E2 -8528.425} C_VEL
LIN {X 0,Y 565.41,Z 782.698,A -85,B 0,C 180,E1 -8530.151,E2 -8530.151} C_VEL
LIN {X 0,Y 564.093,Z 797.426,A -85,B 0,C 180,E1 -8531.929,E2 -8531.929} C_VEL
LIN {X 0,Y 563.035,Z 810.018,A -85,B 0,C 180,E1 -8533.704,E2 -8533.704} C_VEL
LIN {X 0,Y 562.119,Z 821.97,A -85,B 0,C 180,E1 -8535.685,E2 -8535.685} C_VEL
LIN {X 0,Y 561.447,Z 831.988,A -85,B 0,C 180,E1 -8537.66,E2 -8537.66} C_VEL
LIN {X 0,Y 560.944,Z 840.537,A -85,B 0,C 180,E1 -8539.732,E2 -8539.732} C_VEL
LIN {X 0,Y 560.624,Z 847.453,A -85,B 0,C 180,E1 -8541.836,E2 -8541.836} C_VEL
LIN {X 0,Y 560.454,Z 852.782,A -85,B 0,C 180,E1 -8543.958,E2 -8543.958} C_VEL
LIN {X 0,Y 560.369,Z 856.537,A -85,B 0,C 180,E1 -8546.112,E2 -8546.112} C_VEL
LIN {X 0,Y 560.329,Z 858.601,A -85,B 0,C 180,E1 -8548.262,E2 -8548.262} C_VEL
LIN {X 0,Y 560.312,Z 859.114,A -85,B 0,C 180,E1 -8550.511,E2 -8550.511} C_VEL
LIN {X 0,Y 560.337,Z 858.029,A -85,B 0,C 180,E1 -8552.659,E2 -8552.659} C_VEL
LIN {X 0,Y 560.397,Z 855.253,A -85,B 0,C 180,E1 -8554.81,E2 -8554.81} C_VEL
LIN {X 0,Y 560.497,Z 850.869,A -85,B 0,C 180,E1 -8556.968,E2 -8556.968} C_VEL
LIN {X 0,Y 560.721,Z 845.146,A -85,B 0,C 180,E1 -8559.028,E2 -8559.028} C_VEL
LIN {X 0,Y 561.142,Z 837.294,A -85,B 0,C 180,E1 -8561.199,E2 -8561.199} C_VEL
LIN {X 0,Y 561.66,Z 828.399,A -85,B 0,C 180,E1 -8563.172,E2 -8563.172} C_VEL
LIN {X 0,Y 562.475,Z 817.104,A -85,B 0,C 180,E1 -8565.254,E2 -8565.254} C_VEL
LIN {X 0,Y 563.456,Z 804.985,A -85,B 0,C 180,E1 -8567.132,E2 -8567.132} C_VEL
LIN {X 0,Y 564.689,Z 790.849,A -85,B 0,C 180,E1 -8568.994,E2 -8568.994} C_VEL
LIN {X 0,Y 566.137,Z 774.706,A -85,B 0,C 180,E1 -8570.793,E2 -8570.793} C_VEL
LIN {X 0,Y 567.626,Z 758.103,A -85,B 0,C 180,E1 -8572.364,E2 -8572.364} C_VEL
LIN {X 0,Y 569.15,Z 740.648,A -85,B 0,C 180,E1 -8573.778,E2 -8573.778} C_VEL
LIN {X 0,Y 570.738,Z 721.654,A -85,B 0,C 180,E1 -8575.085,E2 -8575.085} C_VEL
LIN {X 0,Y 572.175,Z 702.773,A -85,B 0,C 180,E1 -8576.184,E2 -8576.184} C_VEL
LIN {X 0,Y 573.627,Z 681.462,A -85,B 0,C 180,E1 -8577.205,E2 -8577.205} C_VEL
LIN {X 0,Y 574.813,Z 660.27,A -85,B 0,C 180,E1 -8578.013,E2 -8578.013} C_VEL
LIN {X 0,Y 575.742,Z 638.56,A -85,B 0,C 180,E1 -8578.652,E2 -8578.652} C_VEL
LIN {X 0,Y 576.652,Z 611.573,A -85,B 0,C 180,E1 -8579.22,E2 -8579.22} C_VEL
LIN {X 0,Y 580.684,Z 509.281,A -85,B 0,C 180,E1 -8581.008,E2 -8581.008} C_VEL
LIN {X 0,Y 583.434,Z 425.67,A -85,B 0,C 180,E1 -8582.304,E2 -8582.304} C_VEL
LIN {X 0,Y 585.388,Z 345.041,A -85,B 0,C 180,E1 -8583.426,E2 -8583.426} C_VEL
LIN {X 0,Y 586.453,Z 339.732,A -85,B 0,C 180,E1 -8583.65,E2 -8583.65} C_VEL
LIN {X 0,Y 586.414,Z 308.226,A -85,B 0,C 180,E1 -8585.745,E2 -8585.745} C_VEL
LIN {X 0,Y 587.241,Z 275.669,A -85,B 0,C 180,E1 -8588.083,E2 -8588.083} C_VEL
LIN {X 0,Y 578.615,Z 253.002,A -85,B 0,C 180,E1 -8590.523,E2 -8590.523} C_VEL
LIN {X 0,Y 570.838,Z 235.075,A -85,B 0,C 180,E1 -8592.487,E2 -8592.487} C_VEL
LIN {X 0,Y 562.953,Z 219.066,A -85,B 0,C 180,E1 -8594.292,E2 -8594.292} C_VEL
LIN {X 0,Y 561.477,Z 215.608,A -85,B 0,C 180,E1 -8594.655,E2 -8594.655} C_VEL
LIN {X 0,Y 561.429,Z 215.301,A -85,B 0,C 180,E1 -8594.715,E2 -8594.715} C_VEL
LIN {X 0,Y 561.439,Z 215.303,A -85,B 0,C 180,E1 -8597.961,E2 -8597.961} C_VEL
LIN {X 0,Y 561.422,Z 215.3,A -85,B 0,C 180,E1 -8601.268,E2 -8601.268} C_VEL
LIN {X 0,Y 561.438,Z 215.294,A -85,B 0,C 180,E1 -8604.654,E2 -8604.654} C_VEL
LIN {X 0,Y 561.435,Z 215.283,A -85,B 0,C 180,E1 -8607.966,E2 -8607.966} C_VEL
LIN {X 0,Y 561.425,Z 215.277,A -85,B 0,C 180,E1 -8611.258,E2 -8611.258} C_VEL
LIN {X 0,Y 561.438,Z 215.29,A -85,B 0,C 180,E1 -8614.583,E2 -8614.583} C_VEL
LIN {X 0,Y 561.437,Z 215.282,A -85,B 0,C 180,E1 -8617.927,E2 -8617.927} C_VEL
LIN {X 0,Y 561.428,Z 215.272,A -85,B 0,C 180,E1 -8621.302,E2 -8621.302} C_VEL
LIN {X 0,Y 561.433,Z 215.291,A -85,B 0,C 180,E1 -8624.611,E2 -8624.611} C_VEL
LIN {X 0,Y 561.428,Z 215.266,A -85,B 0,C 180,E1 -8627.973,E2 -8627.973} C_VEL
LIN {X 0,Y 561.435,Z 215.294,A -85,B 0,C 180,E1 -8631.293,E2 -8631.293} C_VEL
LIN {X 0,Y 561.418,Z 215.268,A -85,B 0,C 180,E1 -8634.481,E2 -8634.481} C_VEL
LIN {X 0,Y 561.435,Z 215.295,A -85,B 0,C 180,E1 -8637.857,E2 -8637.857} C_VEL
LIN {X 0,Y 561.438,Z 215.263,A -85,B 0,C 180,E1 -8641.225,E2 -8641.225} C_VEL
LIN {X 0,Y 561.415,Z 215.293,A -85,B 0,C 180,E1 -8644.495,E2 -8644.495} C_VEL
LIN {X 0,Y 561.434,Z 215.265,A -85,B 0,C 180,E1 -8647.882,E2 -8647.882} C_VEL
LIN {X 0,Y 561.439,Z 215.293,A -85,B 0,C 180,E1 -8651.194,E2 -8651.194} C_VEL
LIN {X 0,Y 561.411,Z 215.294,A -85,B 0,C 180,E1 -8654.439,E2 -8654.439} C_VEL
LIN {X 0,Y 561.441,Z 215.295,A -85,B 0,C 180,E1 -8657.731,E2 -8657.731} C_VEL
LIN {X 0,Y 561.428,Z 215.292,A -85,B 0,C 180,E1 -8661.085,E2 -8661.085} C_VEL
LIN {X 0,Y 561.406,Z 215.294,A -85,B 0,C 180,E1 -8664.406,E2 -8664.406} C_VEL
LIN {X 0,Y 561.447,Z 215.292,A -85,B 0,C 180,E1 -8667.734,E2 -8667.734} C_VEL
LIN {X 0,Y 561.411,Z 215.298,A -85,B 0,C 180,E1 -8670.979,E2 -8670.979} C_VEL
LIN {X 0,Y 561.404,Z 215.296,A -85,B 0,C 180,E1 -8674.374,E2 -8674.374} C_VEL
LIN {X 0,Y 561.462,Z 215.418,A -85,B 0,C 180,E1 -8677.632,E2 -8677.632} C_VEL
LIN {X 0,Y 562.826,Z 218.91,A -85,B 0,C 180,E1 -8678.059,E2 -8678.059} C_VEL
LIN {X 0,Y 563.963,Z 221.123,A -85,B 0,C 180,E1 -8678.356,E2 -8678.356} C_VEL
LIN {X 0,Y 570.911,Z 234.738,A -85,B 0,C 180,E1 -8680.129,E2 -8680.129} C_VEL
LIN {X 0,Y 580.547,Z 253.699,A -85,B 0,C 180,E1 -8682.466,E2 -8682.466} C_VEL
LIN {X 0,Y 592.791,Z 278.925,A -85,B 0,C 180,E1 -8685.302,E2 -8685.302} C_VEL
LIN {X 0,Y 594.513,Z 283.316,A -85,B 0,C 180,E1 -8685.735,E2 -8685.735} C_VEL
LIN {X 0,Y 592.128,Z 310.199,A -85,B 0,C 180,E1 -8687.251,E2 -8687.251} C_VEL
LIN {X 0,Y 594.916,Z 334.019,A -85,B 0,C 180,E1 -8687.851,E2 -8687.851} C_VEL
LIN {X 0,Y 588.562,Z 580.572,A -85,B 0,C 180,E1 -8691.348,E2 -8691.348} C_VEL
LIN {X 0,Y 586.04,Z 692.74,A -85,B 0,C 180,E1 -8692.903,E2 -8692.903} C_VEL
LIN {X 0,Y 584.879,Z 717.274,A -85,B 0,C 180,E1 -8693.409,E2 -8693.409} C_VEL
LIN {X 0,Y 583.511,Z 739.8,A -85,B 0,C 180,E1 -8694.025,E2 -8694.025} C_VEL
LIN {X 0,Y 581.762,Z 763.298,A -85,B 0,C 180,E1 -8694.846,E2 -8694.846} C_VEL
LIN {X 0,Y 579.948,Z 784.469,A -85,B 0,C 180,E1 -8695.742,E2 -8695.742} C_VEL
LIN {X 0,Y 577.776,Z 807.376,A -85,B 0,C 180,E1 -8696.907,E2 -8696.907} C_VEL
LIN {X 0,Y 575.695,Z 827.837,A -85,B 0,C 180,E1 -8698.13,E2 -8698.13} C_VEL
LIN {X 0,Y 573.372,Z 849.27,A -85,B 0,C 180,E1 -8699.621,E2 -8699.621} C_VEL
LIN {X 0,Y 571.381,Z 867.088,A -85,B 0,C 180,E1 -8701.043,E2 -8701.043} C_VEL
LIN {X 0,Y 569.065,Z 887.627,A -85,B 0,C 180,E1 -8702.93,E2 -8702.93} C_VEL
LIN {X 0,Y 567.25,Z 903.878,A -85,B 0,C 180,E1 -8704.638,E2 -8704.638} C_VEL
LIN {X 0,Y 565.359,Z 921.592,A -85,B 0,C 180,E1 -8706.772,E2 -8706.772} C_VEL
LIN {X 0,Y 563.946,Z 935.489,A -85,B 0,C 180,E1 -8708.687,E2 -8708.687} C_VEL
LIN {X 0,Y 562.613,Z 950.16,A -85,B 0,C 180,E1 -8711.02,E2 -8711.02} C_VEL
LIN {X 0,Y 561.737,Z 961.076,A -85,B 0,C 180,E1 -8713.027,E2 -8713.027} C_VEL
LIN {X 0,Y 560.971,Z 972.316,A -85,B 0,C 180,E1 -8715.444,E2 -8715.444} C_VEL
LIN {X 0,Y 560.518,Z 980.454,A -85,B 0,C 180,E1 -8717.535,E2 -8717.535} C_VEL
LIN {X 0,Y 560.186,Z 988.207,A -85,B 0,C 180,E1 -8719.926,E2 -8719.926} C_VEL
LIN {X 0,Y 559.997,Z 993.849,A -85,B 0,C 180,E1 -8722.201,E2 -8722.201} C_VEL
LIN {X 0,Y 559.936,Z 997.751,A -85,B 0,C 180,E1 -8724.261,E2 -8724.261} C_VEL
LIN {X 0,Y 559.901,Z 1000.905,A -85,B 0,C 180,E1 -8726.724,E2 -8726.724} C_VEL
LIN {X 0,Y 559.899,Z 1002.184,A -85,B 0,C 180,E1 -8728.977,E2 -8728.977} C_VEL
LIN {X 0,Y 559.894,Z 1002.207,A -85,B 0,C 180,E1 -8730.921,E2 -8730.921} C_VEL
LIN {X 0,Y 559.891,Z 1001.05,A -85,B 0,C 180,E1 -8733.071,E2 -8733.071} C_VEL
LIN {X 0,Y 559.921,Z 998.071,A -85,B 0,C 180,E1 -8735.534,E2 -8735.534} C_VEL
LIN {X 0,Y 559.985,Z 994.242,A -85,B 0,C 180,E1 -8737.593,E2 -8737.593} C_VEL
LIN {X 0,Y 560.164,Z 989.198,A -85,B 0,C 180,E1 -8739.659,E2 -8739.659} C_VEL
LIN {X 0,Y 560.469,Z 981.347,A -85,B 0,C 180,E1 -8742.153,E2 -8742.153} C_VEL
LIN {X 0,Y 560.892,Z 973.239,A -85,B 0,C 180,E1 -8744.242,E2 -8744.242} C_VEL
LIN {X 0,Y 561.577,Z 962.61,A -85,B 0,C 180,E1 -8746.552,E2 -8746.552} C_VEL
LIN {X 0,Y 562.482,Z 950.414,A -85,B 0,C 180,E1 -8748.769,E2 -8748.769} C_VEL
LIN {X 0,Y 563.614,Z 936.977,A -85,B 0,C 180,E1 -8750.891,E2 -8750.891} C_VEL
LIN {X 0,Y 564.998,Z 922.006,A -85,B 0,C 180,E1 -8752.913,E2 -8752.913} C_VEL
LIN {X 0,Y 566.588,Z 905.371,A -85,B 0,C 180,E1 -8754.894,E2 -8754.894} C_VEL
LIN {X 0,Y 568.331,Z 887.591,A -85,B 0,C 180,E1 -8756.713,E2 -8756.713} C_VEL
LIN {X 0,Y 570.202,Z 868.597,A -85,B 0,C 180,E1 -8758.431,E2 -8758.431} C_VEL
LIN {X 0,Y 572.135,Z 848.552,A -85,B 0,C 180,E1 -8759.989,E2 -8759.989} C_VEL
LIN {X 0,Y 574.143,Z 827.442,A -85,B 0,C 180,E1 -8761.421,E2 -8761.421} C_VEL
LIN {X 0,Y 575.917,Z 806.696,A -85,B 0,C 180,E1 -8762.627,E2 -8762.627} C_VEL
LIN {X 0,Y 577.801,Z 783.543,A -85,B 0,C 180,E1 -8763.778,E2 -8763.778} C_VEL
LIN {X 0,Y 579.366,Z 761.816,A -85,B 0,C 180,E1 -8764.67,E2 -8764.67} C_VEL
LIN {X 0,Y 580.894,Z 737.63,A -85,B 0,C 180,E1 -8765.487,E2 -8765.487} C_VEL
LIN {X 0,Y 582,Z 715.071,A -85,B 0,C 180,E1 -8766.076,E2 -8766.076} C_VEL
LIN {X 0,Y 582.938,Z 690.138,A -85,B 0,C 180,E1 -8766.559,E2 -8766.559} C_VEL
LIN {X 0,Y 585.654,Z 533.304,A -85,B 0,C 180,E1 -8768.652,E2 -8768.652} C_VEL
LIN {X 0,Y 588.603,Z 421.987,A -85,B 0,C 180,E1 -8770.301,E2 -8770.301} C_VEL
LIN {X 0,Y 592.073,Z 331.436,A -85,B 0,C 180,E1 -8771.777,E2 -8771.777} C_VEL
LIN {X 0,Y 592.101,Z 329.405,A -85,B 0,C 180,E1 -8771.864,E2 -8771.864} C_VEL
LIN {X 0,Y 597.294,Z 307.596,A -85,B 0,C 180,E1 -8773.474,E2 -8773.474} C_VEL
LIN {X 0,Y 602.859,Z 290.39,A -85,B 0,C 180,E1 -8774.863,E2 -8774.863} C_VEL
LIN {X 0,Y 601.971,Z 285.99,A -85,B 0,C 180,E1 -8776.028,E2 -8776.028} C_VEL
LIN {X 0,Y 601.511,Z 283.922,A -85,B 0,C 180,E1 -8776.905,E2 -8776.905} C_VEL
LIN {X 0,Y 601.513,Z 282.186,A -85,B 0,C 180,E1 -8778.196,E2 -8778.196} C_VEL
LIN {X 0,Y 601.236,Z 284.033,A -85,B 0,C 180,E1 -8779.689,E2 -8779.689} C_VEL
LIN {X 0,Y 601.422,Z 287.216,A -85,B 0,C 180,E1 -8780.819,E2 -8780.819} C_VEL
LIN {X 0,Y 601.421,Z 288.711,A -85,B 0,C 180,E1 -8781.187,E2 -8781.187} C_VEL
LIN {X 0,Y 594.149,Z 309.834,A -85,B 0,C 180,E1 -8783.194,E2 -8783.194} C_VEL
LIN {X 0,Y 587.473,Z 337.328,A -85,B 0,C 180,E1 -8785.593,E2 -8785.593} C_VEL
LIN {X 0,Y 581.912,Z 370.482,A -85,B 0,C 180,E1 -8788.278,E2 -8788.278} C_VEL
LIN {X 0,Y 576.869,Z 412.068,A -85,B 0,C 180,E1 -8791.419,E2 -8791.419} C_VEL
LIN {X 0,Y 576.6,Z 416.359,A -85,B 0,C 180,E1 -8791.703,E2 -8791.703} C_VEL
LIN {X 0,Y 579.297,Z 444.577,A -85,B 0,C 180,E1 -8792.867,E2 -8792.867} C_VEL
LIN {X 0,Y 581.891,Z 479.086,A -85,B 0,C 180,E1 -8794.101,E2 -8794.101} C_VEL
LIN {X 0,Y 582.738,Z 496.873,A -85,B 0,C 180,E1 -8794.649,E2 -8794.649} C_VEL
LIN {X 0,Y 575.952,Z 603.696,A -85,B 0,C 180,E1 -8796.838,E2 -8796.838} C_VEL
LIN {X 0,Y 571.963,Z 688.572,A -85,B 0,C 180,E1 -8798.526,E2 -8798.526} C_VEL
LIN {X 0,Y 570.83,Z 711.243,A -85,B 0,C 180,E1 -8799.176,E2 -8799.176} C_VEL
LIN {X 0,Y 569.701,Z 732.552,A -85,B 0,C 180,E1 -8799.986,E2 -8799.986} C_VEL
LIN {X 0,Y 568.545,Z 752.867,A -85,B 0,C 180,E1 -8800.959,E2 -8800.959} C_VEL
LIN {X 0,Y 567.462,Z 771.005,A -85,B 0,C 180,E1 -8802.04,E2 -8802.04} C_VEL
LIN {X 0,Y 566.378,Z 788.148,A -85,B 0,C 180,E1 -8803.276,E2 -8803.276} C_VEL
LIN {X 0,Y 565.418,Z 802.733,A -85,B 0,C 180,E1 -8804.533,E2 -8804.533} C_VEL
LIN {X 0,Y 564.477,Z 816.474,A -85,B 0,C 180,E1 -8805.955,E2 -8805.955} C_VEL
LIN {X 0,Y 563.63,Z 828.893,A -85,B 0,C 180,E1 -8807.5,E2 -8807.5} C_VEL
LIN {X 0,Y 562.93,Z 839.125,A -85,B 0,C 180,E1 -8809.044,E2 -8809.044} C_VEL
LIN {X 0,Y 562.29,Z 848.446,A -85,B 0,C 180,E1 -8810.791,E2 -8810.791} C_VEL
LIN {X 0,Y 561.818,Z 855.758,A -85,B 0,C 180,E1 -8812.535,E2 -8812.535} C_VEL
LIN {X 0,Y 561.465,Z 861.497,A -85,B 0,C 180,E1 -8814.379,E2 -8814.379} C_VEL
LIN {X 0,Y 561.197,Z 865.371,A -85,B 0,C 180,E1 -8816.22,E2 -8816.22} C_VEL
LIN {X 0,Y 561.012,Z 867.549,A -85,B 0,C 180,E1 -8818.162,E2 -8818.162} C_VEL
LIN {X 0,Y 560.919,Z 867.885,A -85,B 0,C 180,E1 -8820,E2 -8820} C_VEL
LIN {X 0,Y 560.867,Z 866.419,A -85,B 0,C 180,E1 -8821.941,E2 -8821.941} C_VEL
LIN {X 0,Y 560.893,Z 863.09,A -85,B 0,C 180,E1 -8823.884,E2 -8823.884} C_VEL
LIN {X 0,Y 561.01,Z 858.171,A -85,B 0,C 180,E1 -8825.728,E2 -8825.728} C_VEL
LIN {X 0,Y 561.215,Z 851.408,A -85,B 0,C 180,E1 -8827.576,E2 -8827.576} C_VEL
LIN {X 0,Y 561.545,Z 843.168,A -85,B 0,C 180,E1 -8829.325,E2 -8829.325} C_VEL
LIN {X 0,Y 562.042,Z 832.882,A -85,B 0,C 180,E1 -8831.077,E2 -8831.077} C_VEL
LIN {X 0,Y 562.681,Z 821.036,A -85,B 0,C 180,E1 -8832.73,E2 -8832.73} C_VEL
LIN {X 0,Y 563.459,Z 807.62,A -85,B 0,C 180,E1 -8834.28,E2 -8834.28} C_VEL
LIN {X 0,Y 564.359,Z 792.576,A -85,B 0,C 180,E1 -8835.728,E2 -8835.728} C_VEL
LIN {X 0,Y 565.367,Z 775.732,A -85,B 0,C 180,E1 -8837.073,E2 -8837.073} C_VEL
LIN {X 0,Y 566.359,Z 758.188,A -85,B 0,C 180,E1 -8838.227,E2 -8838.227} C_VEL
LIN {X 0,Y 567.343,Z 740.261,A -85,B 0,C 180,E1 -8839.189,E2 -8839.189} C_VEL
LIN {X 0,Y 568.303,Z 720.779,A -85,B 0,C 180,E1 -8840.026,E2 -8840.026} C_VEL
LIN {X 0,Y 569.15,Z 700.322,A -85,B 0,C 180,E1 -8840.693,E2 -8840.693} C_VEL
LIN {X 0,Y 569.857,Z 679.643,A -85,B 0,C 180,E1 -8841.166,E2 -8841.166} C_VEL
LIN {X 0,Y 574.449,Z 491.167,A -85,B 0,C 180,E1 -8844.104,E2 -8844.104} C_VEL
LIN {X 0,Y 570.367,Z 454.133,A -85,B 0,C 180,E1 -8844.937,E2 -8844.937} C_VEL
LIN {X 0,Y 573.177,Z 401.497,A -85,B 0,C 180,E1 -8848.384,E2 -8848.384} C_VEL
LIN {X 0,Y 576.239,Z 350.111,A -85,B 0,C 180,E1 -8851.79,E2 -8851.79} C_VEL
LIN {X 0,Y 579.604,Z 298.699,A -85,B 0,C 180,E1 -8855.244,E2 -8855.244} C_VEL
LIN {X 0,Y 581.653,Z 266.917,A -85,B 0,C 180,E1 -8857.42,E2 -8857.42} C_VEL
LIN {X 0,Y 573.104,Z 244.424,A -85,B 0,C 180,E1 -8859.699,E2 -8859.699} C_VEL
LIN {X 0,Y 564.311,Z 222.551,A -85,B 0,C 180,E1 -8862.062,E2 -8862.062} C_VEL
LIN {X 0,Y 563.532,Z 221.076,A -85,B 0,C 180,E1 -8862.24,E2 -8862.24} C_VEL
LIN {X 0,Y 561.352,Z 218.415,A -85,B 0,C 180,E1 -8862.655,E2 -8862.655} C_VEL
LIN {X 0,Y 557.652,Z 216.768,A -85,B 0,C 180,E1 -8863.235,E2 -8863.235} C_VEL
LIN {X 0,Y 554.482,Z 216.314,A -85,B 0,C 180,E1 -8863.876,E2 -8863.876} C_VEL
LIN {X 0,Y 553.485,Z 216.285,A -85,B 0,C 180,E1 -8864.422,E2 -8864.422} C_VEL
LIN {X 0,Y 553.521,Z 216.448,A -85,B 0,C 180,E1 -8864.724,E2 -8864.724} C_VEL
LIN {X 0,Y 554.89,Z 219.882,A -85,B 0,C 180,E1 -8865.087,E2 -8865.087} C_VEL
LIN {X 0,Y 555.954,Z 221.762,A -85,B 0,C 180,E1 -8865.314,E2 -8865.314} C_VEL
LIN {X 0,Y 563.877,Z 237.896,A -85,B 0,C 180,E1 -8867.159,E2 -8867.159} C_VEL
LIN {X 0,Y 571.245,Z 254.839,A -85,B 0,C 180,E1 -8869.051,E2 -8869.051} C_VEL
LIN {X 0,Y 579.569,Z 276.454,A -85,B 0,C 180,E1 -8871.401,E2 -8871.401} C_VEL
LIN {X 0,Y 580.664,Z 279.683,A -85,B 0,C 180,E1 -8871.742,E2 -8871.742} C_VEL
LIN {X 0,Y 579.819,Z 321.696,A -85,B 0,C 180,E1 -8874.711,E2 -8874.711} C_VEL
LIN {X 0,Y 579.92,Z 342.208,A -85,B 0,C 180,E1 -8876.038,E2 -8876.038} C_VEL
LIN {X 0,Y 578.554,Z 349.119,A -85,B 0,C 180,E1 -8876.292,E2 -8876.292} C_VEL
LIN {X 0,Y 576.214,Z 442.69,A -85,B 0,C 180,E1 -8877.602,E2 -8877.602} C_VEL
LIN {X 0,Y 573.102,Z 528.948,A -85,B 0,C 180,E1 -8878.994,E2 -8878.994} C_VEL
LIN {X 0,Y 569.13,Z 626.101,A -85,B 0,C 180,E1 -8880.767,E2 -8880.767} C_VEL
LIN {X 0,Y 568.324,Z 648.408,A -85,B 0,C 180,E1 -8881.317,E2 -8881.317} C_VEL
LIN {X 0,Y 567.159,Z 670.619,A -85,B 0,C 180,E1 -8882.062,E2 -8882.062} C_VEL
LIN {X 0,Y 565.851,Z 691.3,A -85,B 0,C 180,E1 -8882.949,E2 -8882.949} C_VEL
LIN {X 0,Y 564.367,Z 711.189,A -85,B 0,C 180,E1 -8883.992,E2 -8883.992} C_VEL
LIN {X 0,Y 562.705,Z 731.31,A -85,B 0,C 180,E1 -8885.262,E2 -8885.262} C_VEL
LIN {X 0,Y 561.058,Z 749.599,A -85,B 0,C 180,E1 -8886.633,E2 -8886.633} C_VEL
LIN {X 0,Y 559.43,Z 767.104,A -85,B 0,C 180,E1 -8888.175,E2 -8888.175} C_VEL
LIN {X 0,Y 557.857,Z 783.435,A -85,B 0,C 180,E1 -8889.871,E2 -8889.871} C_VEL
LIN {X 0,Y 556.535,Z 797.387,A -85,B 0,C 180,E1 -8891.566,E2 -8891.566} C_VEL
LIN {X 0,Y 555.334,Z 810.837,A -85,B 0,C 180,E1 -8893.472,E2 -8893.472} C_VEL
LIN {X 0,Y 554.391,Z 822.259,A -85,B 0,C 180,E1 -8895.374,E2 -8895.374} C_VEL
LIN {X 0,Y 553.621,Z 832.861,A -85,B 0,C 180,E1 -8897.483,E2 -8897.483} C_VEL
LIN {X 0,Y 553.078,Z 841.431,A -85,B 0,C 180,E1 -8899.584,E2 -8899.584} C_VEL
LIN {X 0,Y 552.731,Z 848.333,A -85,B 0,C 180,E1 -8901.701,E2 -8901.701} C_VEL
LIN {X 0,Y 552.538,Z 853.742,A -85,B 0,C 180,E1 -8903.871,E2 -8903.871} C_VEL
LIN {X 0,Y 552.438,Z 857.514,A -85,B 0,C 180,E1 -8906.056,E2 -8906.056} C_VEL
LIN {X 0,Y 552.394,Z 859.597,A -85,B 0,C 180,E1 -8908.237,E2 -8908.237} C_VEL
LIN {X 0,Y 552.374,Z 860.115,A -85,B 0,C 180,E1 -8910.519,E2 -8910.519} C_VEL
LIN {X 0,Y 552.403,Z 859.016,A -85,B 0,C 180,E1 -8912.697,E2 -8912.697} C_VEL
LIN {X 0,Y 552.47,Z 856.226,A -85,B 0,C 180,E1 -8914.88,E2 -8914.88} C_VEL
LIN {X 0,Y 552.584,Z 851.812,A -85,B 0,C 180,E1 -8917.068,E2 -8917.068} C_VEL
LIN {X 0,Y 552.848,Z 845.705,A -85,B 0,C 180,E1 -8919.263,E2 -8919.263} C_VEL
LIN {X 0,Y 553.292,Z 838.188,A -85,B 0,C 180,E1 -8921.36,E2 -8921.36} C_VEL
LIN {X 0,Y 553.898,Z 828.756,A -85,B 0,C 180,E1 -8923.466,E2 -8923.466} C_VEL
LIN {X 0,Y 554.737,Z 817.93,A -85,B 0,C 180,E1 -8925.472,E2 -8925.472} C_VEL
LIN {X 0,Y 555.845,Z 805.023,A -85,B 0,C 180,E1 -8927.482,E2 -8927.482} C_VEL
LIN {X 0,Y 557.108,Z 791.427,A -85,B 0,C 180,E1 -8929.283,E2 -8929.283} C_VEL
LIN {X 0,Y 558.588,Z 775.957,A -85,B 0,C 180,E1 -8931.033,E2 -8931.033} C_VEL
LIN {X 0,Y 560.214,Z 758.821,A -85,B 0,C 180,E1 -8932.676,E2 -8932.676} C_VEL
LIN {X 0,Y 561.811,Z 741.377,A -85,B 0,C 180,E1 -8934.102,E2 -8934.102} C_VEL
LIN {X 0,Y 563.487,Z 722.246,A -85,B 0,C 180,E1 -8935.431,E2 -8935.431} C_VEL
LIN {X 0,Y 565.053,Z 702.232,A -85,B 0,C 180,E1 -8936.596,E2 -8936.596} C_VEL
LIN {X 0,Y 566.461,Z 682.502,A -85,B 0,C 180,E1 -8937.547,E2 -8937.547} C_VEL
LIN {X 0,Y 567.706,Z 661.32,A -85,B 0,C 180,E1 -8938.366,E2 -8938.366} C_VEL
LIN {X 0,Y 568.667,Z 639.573,A -85,B 0,C 180,E1 -8939.014,E2 -8939.014} C_VEL
LIN {X 0,Y 569.618,Z 612.327,A -85,B 0,C 180,E1 -8939.595,E2 -8939.595} C_VEL
LIN {X 0,Y 573.742,Z 513.351,A -85,B 0,C 180,E1 -8941.363,E2 -8941.363} C_VEL
LIN {X 0,Y 576.593,Z 431.128,A -85,B 0,C 180,E1 -8942.661,E2 -8942.661} C_VEL
LIN {X 0,Y 578.708,Z 347.779,A -85,B 0,C 180,E1 -8943.834,E2 -8943.834} C_VEL
LIN {X 0,Y 580.002,Z 341.168,A -85,B 0,C 180,E1 -8944.116,E2 -8944.116} C_VEL
LIN {X 0,Y 579.996,Z 308.239,A -85,B 0,C 180,E1 -8946.312,E2 -8946.312} C_VEL
LIN {X 0,Y 580.613,Z 279.112,A -85,B 0,C 180,E1 -8948.411,E2 -8948.411} C_VEL
LIN {X 0,Y 572.14,Z 256.868,A -85,B 0,C 180,E1 -8950.823,E2 -8950.823} C_VEL
LIN {X 0,Y 564.396,Z 238.99,A -85,B 0,C 180,E1 -8952.824,E2 -8952.824} C_VEL
LIN {X 0,Y 557.007,Z 223.955,A -85,B 0,C 180,E1 -8954.548,E2 -8954.548} C_VEL
LIN {X 0,Y 555.267,Z 220.416,A -85,B 0,C 180,E1 -8954.952,E2 -8954.952} C_VEL
LIN {X 0,Y 553.664,Z 217.25,A -85,B 0,C 180,E1 -8955.316,E2 -8955.316} C_VEL
LIN {X 0,Y 553.487,Z 216.285,A -85,B 0,C 180,E1 -8955.419,E2 -8955.419} C_VEL
LIN {X 0,Y 553.485,Z 216.28,A -85,B 0,C 180,E1 -8958.884,E2 -8958.884} C_VEL
LIN {X 0,Y 553.497,Z 216.278,A -85,B 0,C 180,E1 -8962.133,E2 -8962.133} C_VEL
LIN {X 0,Y 553.49,Z 216.287,A -85,B 0,C 180,E1 -8965.464,E2 -8965.464} C_VEL
LIN {X 0,Y 553.494,Z 216.282,A -85,B 0,C 180,E1 -8968.902,E2 -8968.902} C_VEL
LIN {X 0,Y 553.491,Z 216.267,A -85,B 0,C 180,E1 -8972.22,E2 -8972.22} C_VEL
LIN {X 0,Y 553.496,Z 216.264,A -85,B 0,C 180,E1 -8975.571,E2 -8975.571} C_VEL
LIN {X 0,Y 553.495,Z 216.28,A -85,B 0,C 180,E1 -8979.042,E2 -8979.042} C_VEL
LIN {X 0,Y 553.486,Z 216.257,A -85,B 0,C 180,E1 -8982.332,E2 -8982.332} C_VEL
LIN {X 0,Y 553.502,Z 216.277,A -85,B 0,C 180,E1 -8985.671,E2 -8985.671} C_VEL
LIN {X 0,Y 553.496,Z 216.265,A -85,B 0,C 180,E1 -8989.066,E2 -8989.066} C_VEL
LIN {X 0,Y 553.48,Z 216.271,A -85,B 0,C 180,E1 -8992.422,E2 -8992.422} C_VEL
LIN {X 0,Y 553.495,Z 216.269,A -85,B 0,C 180,E1 -8995.752,E2 -8995.752} C_VEL
LIN {X 0,Y 553.5,Z 216.268,A -85,B 0,C 180,E1 -8999.172,E2 -8999.172} C_VEL
LIN {X 0,Y 553.478,Z 216.281,A -85,B 0,C 180,E1 -9002.528,E2 -9002.528} C_VEL
LIN {X 0,Y 553.494,Z 216.261,A -85,B 0,C 180,E1 -9005.91,E2 -9005.91} C_VEL
LIN {X 0,Y 553.502,Z 216.274,A -85,B 0,C 180,E1 -9009.252,E2 -9009.252} C_VEL
LIN {X 0,Y 553.471,Z 216.285,A -85,B 0,C 180,E1 -9012.521,E2 -9012.521} C_VEL
LIN {X 0,Y 553.501,Z 216.278,A -85,B 0,C 180,E1 -9015.83,E2 -9015.83} C_VEL
LIN {X 0,Y 553.497,Z 216.278,A -85,B 0,C 180,E1 -9019.195,E2 -9019.195} C_VEL
LIN {X 0,Y 553.467,Z 216.289,A -85,B 0,C 180,E1 -9022.52,E2 -9022.52} C_VEL
LIN {X 0,Y 553.499,Z 216.285,A -85,B 0,C 180,E1 -9025.89,E2 -9025.89} C_VEL
LIN {X 0,Y 553.497,Z 216.278,A -85,B 0,C 180,E1 -9029.245,E2 -9029.245} C_VEL
LIN {X 0,Y 553.46,Z 216.291,A -85,B 0,C 180,E1 -9032.573,E2 -9032.573} C_VEL
LIN {X 0,Y 553.501,Z 216.277,A -85,B 0,C 180,E1 -9035.824,E2 -9035.824} C_VEL
LIN {X 0,Y 553.476,Z 216.421,A -85,B 0,C 180,E1 -9036.816,E2 -9036.816} C_VEL
LIN {X 0,Y 554.881,Z 219.897,A -85,B 0,C 180,E1 -9037.263,E2 -9037.263} C_VEL
LIN {X 0,Y 556.036,Z 221.965,A -85,B 0,C 180,E1 -9037.561,E2 -9037.561} C_VEL
LIN {X 0,Y 565.205,Z 240.074,A -85,B 0,C 180,E1 -9039.954,E2 -9039.954} C_VEL
LIN {X 0,Y 575.598,Z 260.783,A -85,B 0,C 180,E1 -9042.512,E2 -9042.512} C_VEL
LIN {X 0,Y 586.882,Z 284.08,A -85,B 0,C 180,E1 -9045.143,E2 -9045.143} C_VEL
LIN {X 0,Y 587.893,Z 286.655,A -85,B 0,C 180,E1 -9045.401,E2 -9045.401} C_VEL
LIN {X 0,Y 585.671,Z 310.899,A -85,B 0,C 180,E1 -9046.778,E2 -9046.778} C_VEL
LIN {X 0,Y 588.469,Z 335.301,A -85,B 0,C 180,E1 -9047.403,E2 -9047.403} C_VEL
LIN {X 0,Y 581.957,Z 573.346,A -85,B 0,C 180,E1 -9050.829,E2 -9050.829} C_VEL
LIN {X 0,Y 579.108,Z 692.876,A -85,B 0,C 180,E1 -9052.51,E2 -9052.51} C_VEL
LIN {X 0,Y 577.898,Z 717.248,A -85,B 0,C 180,E1 -9053.019,E2 -9053.019} C_VEL
LIN {X 0,Y 576.472,Z 739.786,A -85,B 0,C 180,E1 -9053.643,E2 -9053.643} C_VEL
LIN {X 0,Y 574.658,Z 763.111,A -85,B 0,C 180,E1 -9054.468,E2 -9054.468} C_VEL
LIN {X 0,Y 572.77,Z 784.233,A -85,B 0,C 180,E1 -9055.373,E2 -9055.373} C_VEL
LIN {X 0,Y 570.474,Z 807.48,A -85,B 0,C 180,E1 -9056.569,E2 -9056.569} C_VEL
LIN {X 0,Y 568.337,Z 827.671,A -85,B 0,C 180,E1 -9057.787,E2 -9057.787} C_VEL
LIN {X 0,Y 565.924,Z 849.068,A -85,B 0,C 180,E1 -9059.295,E2 -9059.295} C_VEL
LIN {X 0,Y 563.747,Z 867.705,A -85,B 0,C 180,E1 -9060.807,E2 -9060.807} C_VEL
LIN {X 0,Y 561.419,Z 887.384,A -85,B 0,C 180,E1 -9062.645,E2 -9062.645} C_VEL
LIN {X 0,Y 559.602,Z 903.013,A -85,B 0,C 180,E1 -9064.31,E2 -9064.31} C_VEL
LIN {X 0,Y 557.635,Z 920.451,A -85,B 0,C 180,E1 -9066.431,E2 -9066.431} C_VEL
LIN {X 0,Y 556.167,Z 934.394,A -85,B 0,C 180,E1 -9068.374,E2 -9068.374} C_VEL
LIN {X 0,Y 554.754,Z 949.139,A -85,B 0,C 180,E1 -9070.741,E2 -9070.741} C_VEL
LIN {X 0,Y 553.786,Z 960.626,A -85,B 0,C 180,E1 -9072.884,E2 -9072.884} C_VEL
LIN {X 0,Y 553,Z 971.81,A -85,B 0,C 180,E1 -9075.337,E2 -9075.337} C_VEL
LIN {X 0,Y 552.537,Z 979.916,A -85,B 0,C 180,E1 -9077.458,E2 -9077.458} C_VEL
LIN {X 0,Y 552.204,Z 987.598,A -85,B 0,C 180,E1 -9079.884,E2 -9079.884} C_VEL
LIN {X 0,Y 552.019,Z 993.268,A -85,B 0,C 180,E1 -9082.224,E2 -9082.224} C_VEL
LIN {X 0,Y 551.967,Z 997.063,A -85,B 0,C 180,E1 -9084.282,E2 -9084.282} C_VEL
LIN {X 0,Y 551.94,Z 1000.124,A -85,B 0,C 180,E1 -9086.781,E2 -9086.781} C_VEL
LIN {X 0,Y 551.945,Z 1001.33,A -85,B 0,C 180,E1 -9088.962,E2 -9088.962} C_VEL
LIN {X 0,Y 551.947,Z 1001.321,A -85,B 0,C 180,E1 -9091.038,E2 -9091.038} C_VEL
LIN {X 0,Y 551.954,Z 999.888,A -85,B 0,C 180,E1 -9093.469,E2 -9093.469} C_VEL
LIN {X 0,Y 551.991,Z 996.633,A -85,B 0,C 180,E1 -9095.926,E2 -9095.926} C_VEL
LIN {X 0,Y 552.066,Z 992.393,A -85,B 0,C 180,E1 -9098.122,E2 -9098.122} C_VEL
LIN {X 0,Y 552.28,Z 985.766,A -85,B 0,C 180,E1 -9100.642,E2 -9100.642} C_VEL
LIN {X 0,Y 552.616,Z 978.362,A -85,B 0,C 180,E1 -9102.859,E2 -9102.859} C_VEL
LIN {X 0,Y 553.181,Z 968.437,A -85,B 0,C 180,E1 -9105.302,E2 -9105.302} C_VEL
LIN {X 0,Y 553.964,Z 957.45,A -85,B 0,C 180,E1 -9107.544,E2 -9107.544} C_VEL
LIN {X 0,Y 555.052,Z 943.909,A -85,B 0,C 180,E1 -9109.906,E2 -9109.906} C_VEL
LIN {X 0,Y 556.223,Z 930.908,A -85,B 0,C 180,E1 -9111.846,E2 -9111.846} C_VEL
LIN {X 0,Y 557.734,Z 915.298,A -85,B 0,C 180,E1 -9113.902,E2 -9113.902} C_VEL
LIN {X 0,Y 559.464,Z 898.041,A -85,B 0,C 180,E1 -9115.854,E2 -9115.854} C_VEL
LIN {X 0,Y 561.395,Z 879.458,A -85,B 0,C 180,E1 -9117.701,E2 -9117.701} C_VEL
LIN {X 0,Y 563.277,Z 861.157,A -85,B 0,C 180,E1 -9119.28,E2 -9119.28} C_VEL
LIN {X 0,Y 565.361,Z 840.323,A -85,B 0,C 180,E1 -9120.857,E2 -9120.857} C_VEL
LIN {X 0,Y 567.275,Z 820.217,A -85,B 0,C 180,E1 -9122.162,E2 -9122.162} C_VEL
LIN {X 0,Y 569.313,Z 798.034,A -85,B 0,C 180,E1 -9123.409,E2 -9123.409} C_VEL
LIN {X 0,Y 571.068,Z 776.145,A -85,B 0,C 180,E1 -9124.44,E2 -9124.44} C_VEL
LIN {X 0,Y 572.778,Z 752.775,A -85,B 0,C 180,E1 -9125.359,E2 -9125.359} C_VEL
LIN {X 0,Y 574.146,Z 730.177,A -85,B 0,C 180,E1 -9126.069,E2 -9126.069} C_VEL
LIN {X 0,Y 575.44,Z 704.455,A -85,B 0,C 180,E1 -9126.685,E2 -9126.685} C_VEL
LIN {X 0,Y 576.164,Z 682.191,A -85,B 0,C 180,E1 -9127.062,E2 -9127.062} C_VEL
LIN {X 0,Y 578.616,Z 550.242,A -85,B 0,C 180,E1 -9128.851,E2 -9128.851} C_VEL
LIN {X 0,Y 581.652,Z 443.014,A -85,B 0,C 180,E1 -9130.468,E2 -9130.468} C_VEL
LIN {X 0,Y 585.823,Z 345.904,A -85,B 0,C 180,E1 -9132.074,E2 -9132.074} C_VEL
LIN {X 0,Y 586.386,Z 332.55,A -85,B 0,C 180,E1 -9132.325,E2 -9132.325} C_VEL
LIN {X 0,Y 592.083,Z 311.14,A -85,B 0,C 180,E1 -9133.954,E2 -9133.954} C_VEL
LIN {X 0,Y 597.7,Z 295.313,A -85,B 0,C 180,E1 -9135.281,E2 -9135.281} C_VEL
LIN {X 0,Y 597.063,Z 291.289,A -85,B 0,C 180,E1 -9136.504,E2 -9136.504} C_VEL
LIN {X 0,Y 596.806,Z 289.008,A -85,B 0,C 180,E1 -9137.92,E2 -9137.92} C_VEL
LIN {X 0,Y 596.743,Z 288.9,A -85,B 0,C 180,E1 -9138.358,E2 -9138.358} C_VEL
LIN {X 0,Y 596.491,Z 290.948,A -85,B 0,C 180,E1 -9139.806,E2 -9139.806} C_VEL
LIN {X 0,Y 596.557,Z 293.762,A -85,B 0,C 180,E1 -9140.779,E2 -9140.779} C_VEL
LIN {X 0,Y 589.076,Z 313.361,A -85,B 0,C 180,E1 -9142.701,E2 -9142.701} C_VEL
LIN {X 0,Y 582.028,Z 339.205,A -85,B 0,C 180,E1 -9145.031,E2 -9145.031} C_VEL
LIN {X 0,Y 575.944,Z 371.471,A -85,B 0,C 180,E1 -9147.723,E2 -9147.723} C_VEL
LIN {X 0,Y 570.647,Z 410.651,A -85,B 0,C 180,E1 -9150.762,E2 -9150.762} C_VEL
LIN {X 0,Y 570.699,Z 414.084,A -85,B 0,C 180,E1 -9150.948,E2 -9150.948} C_VEL
LIN {X 0,Y 573.177,Z 442.286,A -85,B 0,C 180,E1 -9152.184,E2 -9152.184} C_VEL
LIN {X 0,Y 575.473,Z 475.641,A -85,B 0,C 180,E1 -9153.438,E2 -9153.438} C_VEL
LIN {X 0,Y 576.496,Z 497.783,A -85,B 0,C 180,E1 -9154.162,E2 -9154.162} C_VEL
LIN {X 0,Y 569.301,Z 603.387,A -85,B 0,C 180,E1 -9156.387,E2 -9156.387} C_VEL
LIN {X 0,Y 564.916,Z 688.685,A -85,B 0,C 180,E1 -9158.142,E2 -9158.142} C_VEL
LIN {X 0,Y 563.657,Z 711.807,A -85,B 0,C 180,E1 -9158.822,E2 -9158.822} C_VEL
LIN {X 0,Y 562.504,Z 732.325,A -85,B 0,C 180,E1 -9159.61,E2 -9159.61} C_VEL
LIN {X 0,Y 561.315,Z 751.668,A -85,B 0,C 180,E1 -9160.542,E2 -9160.542} C_VEL
LIN {X 0,Y 560.101,Z 771.034,A -85,B 0,C 180,E1 -9161.688,E2 -9161.688} C_VEL
LIN {X 0,Y 558.939,Z 788.319,A -85,B 0,C 180,E1 -9162.939,E2 -9162.939} C_VEL
LIN {X 0,Y 557.837,Z 803.862,A -85,B 0,C 180,E1 -9164.296,E2 -9164.296} C_VEL
LIN {X 0,Y 556.901,Z 816.943,A -85,B 0,C 180,E1 -9165.654,E2 -9165.654} C_VEL
LIN {X 0,Y 555.979,Z 829.452,A -85,B 0,C 180,E1 -9167.22,E2 -9167.22} C_VEL
LIN {X 0,Y 555.17,Z 840.396,A -85,B 0,C 180,E1 -9168.889,E2 -9168.889} C_VEL
LIN {X 0,Y 554.524,Z 849.241,A -85,B 0,C 180,E1 -9170.556,E2 -9170.556} C_VEL
LIN {X 0,Y 553.997,Z 856.608,A -85,B 0,C 180,E1 -9172.325,E2 -9172.325} C_VEL
LIN {X 0,Y 553.605,Z 862.426,A -85,B 0,C 180,E1 -9174.195,E2 -9174.195} C_VEL
LIN {X 0,Y 553.309,Z 866.365,A -85,B 0,C 180,E1 -9176.062,E2 -9176.062} C_VEL
LIN {X 0,Y 553.114,Z 868.524,A -85,B 0,C 180,E1 -9177.928,E2 -9177.928} C_VEL
LIN {X 0,Y 552.996,Z 868.976,A -85,B 0,C 180,E1 -9179.793,E2 -9179.793} C_VEL
LIN {X 0,Y 552.93,Z 867.747,A -85,B 0,C 180,E1 -9181.658,E2 -9181.658} C_VEL
LIN {X 0,Y 552.943,Z 864.851,A -85,B 0,C 180,E1 -9183.525,E2 -9183.525} C_VEL
LIN {X 0,Y 553.04,Z 860.244,A -85,B 0,C 180,E1 -9185.395,E2 -9185.395} C_VEL
LIN {X 0,Y 553.236,Z 853.821,A -85,B 0,C 180,E1 -9187.268,E2 -9187.268} C_VEL
LIN {X 0,Y 553.552,Z 845.926,A -85,B 0,C 180,E1 -9189.042,E2 -9189.042} C_VEL
LIN {X 0,Y 554.037,Z 836.053,A -85,B 0,C 180,E1 -9190.818,E2 -9190.818} C_VEL
LIN {X 0,Y 554.663,Z 824.668,A -85,B 0,C 180,E1 -9192.493,E2 -9192.493} C_VEL
LIN {X 0,Y 555.429,Z 811.79,A -85,B 0,C 180,E1 -9194.065,E2 -9194.065} C_VEL
LIN {X 0,Y 556.34,Z 797.092,A -85,B 0,C 180,E1 -9195.563,E2 -9195.563} C_VEL
LIN {X 0,Y 557.324,Z 781.393,A -85,B 0,C 180,E1 -9196.897,E2 -9196.897} C_VEL
LIN {X 0,Y 558.345,Z 764.302,A -85,B 0,C 180,E1 -9198.102,E2 -9198.102} C_VEL
LIN {X 0,Y 559.387,Z 746.229,A -85,B 0,C 180,E1 -9199.148,E2 -9199.148} C_VEL
LIN {X 0,Y 560.404,Z 727.196,A -85,B 0,C 180,E1 -9200.034,E2 -9200.034} C_VEL
LIN {X 0,Y 561.312,Z 707.248,A -85,B 0,C 180,E1 -9200.756,E2 -9200.756} C_VEL
LIN {X 0,Y 562.113,Z 686.328,A -85,B 0,C 180,E1 -9201.308,E2 -9201.308} C_VEL
LIN {X 0,Y 562.84,Z 658.287,A -85,B 0,C 180,E1 -9201.789,E2 -9201.789} C_VEL
LIN {X 0,Y 567.175,Z 492.226,A -85,B 0,C 180,E1 -9204.423,E2 -9204.423} C_VEL
LIN {X 0,Y 562.977,Z 452.936,A -85,B 0,C 180,E1 -9205.343,E2 -9205.343} C_VEL
LIN {X 0,Y 566.015,Z 399.396,A -85,B 0,C 180,E1 -9208.891,E2 -9208.891} C_VEL
LIN {X 0,Y 569.239,Z 347.997,A -85,B 0,C 180,E1 -9212.339,E2 -9212.339} C_VEL
LIN {X 0,Y 572.877,Z 295.512,A -85,B 0,C 180,E1 -9215.906,E2 -9215.906} C_VEL
LIN {X 0,Y 574.654,Z 270.17,A -85,B 0,C 180,E1 -9217.656,E2 -9217.656} C_VEL
LIN {X 0,Y 566.144,Z 247.725,A -85,B 0,C 180,E1 -9219.959,E2 -9219.959} C_VEL
LIN {X 0,Y 557.334,Z 226.081,A -85,B 0,C 180,E1 -9222.341,E2 -9222.341} C_VEL
LIN {X 0,Y 553.502,Z 216.282,A -85,B 0,C 180,E1 -9223.462,E2 -9223.462} C_VEL
LIN {X 0,Y 553.485,Z 216.285,A -85,B 0,C 180,E1 -9224.422,E2 -9224.422} C_VEL
LIN {X 0,Y 554.05,Z 216.863,A -85,B 0,C 180,E1 -9224.73,E2 -9224.73} C_VEL
LIN {X 0,Y 555.877,Z 219.571,A -85,B 0,C 180,E1 -9225.163,E2 -9225.163} C_VEL
LIN {X 0,Y 557.069,Z 224.539,A -85,B 0,C 180,E1 -9225.603,E2 -9225.603} C_VEL
LIN {X 0,Y 557.226,Z 232.762,A -85,B 0,C 180,E1 -9226.13,E2 -9226.13} C_VEL
LIN {X 0,Y 557.162,Z 239.787,A -85,B 0,C 180,E1 -9226.631,E2 -9226.631} C_VEL
LIN {X 0,Y 557.809,Z 242.388,A -85,B 0,C 180,E1 -9226.882,E2 -9226.882} C_VEL
LIN {X 0,Y 565.222,Z 259.709,A -85,B 0,C 180,E1 -9228.847,E2 -9228.847} C_VEL
LIN {X 0,Y 573.102,Z 280.2,A -85,B 0,C 180,E1 -9231.091,E2 -9231.091} C_VEL
LIN {X 0,Y 574.177,Z 283.466,A -85,B 0,C 180,E1 -9231.436,E2 -9231.436} C_VEL
LIN {X 0,Y 573.407,Z 324.892,A -85,B 0,C 180,E1 -9234.351,E2 -9234.351} C_VEL
LIN {X 0,Y 573.395,Z 344.327,A -85,B 0,C 180,E1 -9235.598,E2 -9235.598} C_VEL
LIN {X 0,Y 571.91,Z 351.804,A -85,B 0,C 180,E1 -9235.873,E2 -9235.873} C_VEL
LIN {X 0,Y 569.501,Z 444.205,A -85,B 0,C 180,E1 -9237.18,E2 -9237.18} C_VEL
LIN {X 0,Y 566.346,Z 528.179,A -85,B 0,C 180,E1 -9238.553,E2 -9238.553} C_VEL
LIN {X 0,Y 562.151,Z 625.543,A -85,B 0,C 180,E1 -9240.357,E2 -9240.357} C_VEL
LIN {X 0,Y 561.324,Z 647.713,A -85,B 0,C 180,E1 -9240.902,E2 -9240.902} C_VEL
LIN {X 0,Y 560.201,Z 668.926,A -85,B 0,C 180,E1 -9241.603,E2 -9241.603} C_VEL
LIN {X 0,Y 558.83,Z 690.378,A -85,B 0,C 180,E1 -9242.508,E2 -9242.508} C_VEL
LIN {X 0,Y 557.263,Z 710.898,A -85,B 0,C 180,E1 -9243.578,E2 -9243.578} C_VEL
LIN {X 0,Y 555.654,Z 729.737,A -85,B 0,C 180,E1 -9244.756,E2 -9244.756} C_VEL
LIN {X 0,Y 553.907,Z 748.467,A -85,B 0,C 180,E1 -9246.149,E2 -9246.149} C_VEL
LIN {X 0,Y 552.205,Z 765.569,A -85,B 0,C 180,E1 -9247.651,E2 -9247.651} C_VEL
LIN {X 0,Y 550.615,Z 781.323,A -85,B 0,C 180,E1 -9249.264,E2 -9249.264} C_VEL
LIN {X 0,Y 549.096,Z 796.575,A -85,B 0,C 180,E1 -9251.087,E2 -9251.087} C_VEL
LIN {X 0,Y 547.846,Z 809.646,A -85,B 0,C 180,E1 -9252.912,E2 -9252.912} C_VEL
LIN {X 0,Y 546.736,Z 821.984,A -85,B 0,C 180,E1 -9254.948,E2 -9254.948} C_VEL
LIN {X 0,Y 545.887,Z 832.446,A -85,B 0,C 180,E1 -9257.023,E2 -9257.023} C_VEL
LIN {X 0,Y 545.295,Z 841.157,A -85,B 0,C 180,E1 -9259.113,E2 -9259.113} C_VEL
LIN {X 0,Y 544.893,Z 848.325,A -85,B 0,C 180,E1 -9261.239,E2 -9261.239} C_VEL
LIN {X 0,Y 544.655,Z 854.059,A -85,B 0,C 180,E1 -9263.464,E2 -9263.464} C_VEL
LIN {X 0,Y 544.52,Z 858.022,A -85,B 0,C 180,E1 -9265.682,E2 -9265.682} C_VEL
LIN {X 0,Y 544.463,Z 860.459,A -85,B 0,C 180,E1 -9268,E2 -9268} C_VEL
LIN {X 0,Y 544.452,Z 861.183,A -85,B 0,C 180,E1 -9270.21,E2 -9270.21} C_VEL
LIN {X 0,Y 544.46,Z 860.248,A -85,B 0,C 180,E1 -9272.421,E2 -9272.421} C_VEL
LIN {X 0,Y 544.532,Z 857.68,A -85,B 0,C 180,E1 -9274.634,E2 -9274.634} C_VEL
LIN {X 0,Y 544.661,Z 853.521,A -85,B 0,C 180,E1 -9276.853,E2 -9276.853} C_VEL
LIN {X 0,Y 544.921,Z 847.677,A -85,B 0,C 180,E1 -9279.079,E2 -9279.079} C_VEL
LIN {X 0,Y 545.39,Z 839.904,A -85,B 0,C 180,E1 -9281.313,E2 -9281.313} C_VEL
LIN {X 0,Y 545.984,Z 831.159,A -85,B 0,C 180,E1 -9283.341,E2 -9283.341} C_VEL
LIN {X 0,Y 546.898,Z 820.032,A -85,B 0,C 180,E1 -9285.482,E2 -9285.482} C_VEL
LIN {X 0,Y 547.993,Z 808.097,A -85,B 0,C 180,E1 -9287.412,E2 -9287.412} C_VEL
LIN {X 0,Y 549.373,Z 793.988,A -85,B 0,C 180,E1 -9289.345,E2 -9289.345} C_VEL
LIN {X 0,Y 550.946,Z 778.217,A -85,B 0,C 180,E1 -9291.171,E2 -9291.171} C_VEL
LIN {X 0,Y 552.578,Z 761.895,A -85,B 0,C 180,E1 -9292.782,E2 -9292.782} C_VEL
LIN {X 0,Y 554.315,Z 744.086,A -85,B 0,C 180,E1 -9294.285,E2 -9294.285} C_VEL
LIN {X 0,Y 556.041,Z 725.374,A -85,B 0,C 180,E1 -9295.625,E2 -9295.625} C_VEL
LIN {X 0,Y 557.617,Z 706.84,A -85,B 0,C 180,E1 -9296.749,E2 -9296.749} C_VEL
LIN {X 0,Y 559.211,Z 685.417,A -85,B 0,C 180,E1 -9297.819,E2 -9297.819} C_VEL
LIN {X 0,Y 560.53,Z 663.88,A -85,B 0,C 180,E1 -9298.676,E2 -9298.676} C_VEL
LIN {X 0,Y 561.551,Z 642.269,A -85,B 0,C 180,E1 -9299.34,E2 -9299.34} C_VEL
LIN {X 0,Y 562.531,Z 615.38,A -85,B 0,C 180,E1 -9299.936,E2 -9299.936} C_VEL
LIN {X 0,Y 566.732,Z 519.503,A -85,B 0,C 180,E1 -9301.69,E2 -9301.69} C_VEL
LIN {X 0,Y 569.737,Z 437.707,A -85,B 0,C 180,E1 -9303.01,E2 -9303.01} C_VEL
LIN {X 0,Y 572.056,Z 350.5,A -85,B 0,C 180,E1 -9304.251,E2 -9304.251} C_VEL
LIN {X 0,Y 573.59,Z 342.93,A -85,B 0,C 180,E1 -9304.57,E2 -9304.57} C_VEL
LIN {X 0,Y 573.621,Z 308.086,A -85,B 0,C 180,E1 -9306.9,E2 -9306.9} C_VEL
LIN {X 0,Y 574.174,Z 282.895,A -85,B 0,C 180,E1 -9308.724,E2 -9308.724} C_VEL
LIN {X 0,Y 565.522,Z 260.216,A -85,B 0,C 180,E1 -9311.208,E2 -9311.208} C_VEL
LIN {X 0,Y 557.598,Z 241.874,A -85,B 0,C 180,E1 -9313.277,E2 -9313.277} C_VEL
LIN {X 0,Y 549.846,Z 226.072,A -85,B 0,C 180,E1 -9315.124,E2 -9315.124} C_VEL
LIN {X 0,Y 547.147,Z 221.142,A -85,B 0,C 180,E1 -9315.726,E2 -9315.726} C_VEL
LIN {X 0,Y 545.636,Z 217.747,A -85,B 0,C 180,E1 -9316.101,E2 -9316.101} C_VEL
LIN {X 0,Y 545.561,Z 217.262,A -85,B 0,C 180,E1 -9316.148,E2 -9316.148} C_VEL
LIN {X 0,Y 545.556,Z 217.26,A -85,B 0,C 180,E1 -9319.548,E2 -9319.548} C_VEL
LIN {X 0,Y 545.548,Z 217.257,A -85,B 0,C 180,E1 -9322.915,E2 -9322.915} C_VEL
LIN {X 0,Y 545.557,Z 217.259,A -85,B 0,C 180,E1 -9326.313,E2 -9326.313} C_VEL
LIN {X 0,Y 545.571,Z 217.27,A -85,B 0,C 180,E1 -9329.735,E2 -9329.735} C_VEL
LIN {X 0,Y 545.55,Z 217.267,A -85,B 0,C 180,E1 -9333.2,E2 -9333.2} C_VEL
LIN {X 0,Y 545.557,Z 217.242,A -85,B 0,C 180,E1 -9336.564,E2 -9336.564} C_VEL
LIN {X 0,Y 545.555,Z 217.265,A -85,B 0,C 180,E1 -9339.956,E2 -9339.956} C_VEL
LIN {X 0,Y 545.552,Z 217.256,A -85,B 0,C 180,E1 -9343.386,E2 -9343.386} C_VEL
LIN {X 0,Y 545.558,Z 217.251,A -85,B 0,C 180,E1 -9346.756,E2 -9346.756} C_VEL
LIN {X 0,Y 545.548,Z 217.274,A -85,B 0,C 180,E1 -9350.186,E2 -9350.186} C_VEL
LIN {X 0,Y 545.557,Z 217.241,A -85,B 0,C 180,E1 -9353.581,E2 -9353.581} C_VEL
LIN {X 0,Y 545.559,Z 217.27,A -85,B 0,C 180,E1 -9357.058,E2 -9357.058} C_VEL
LIN {X 0,Y 545.535,Z 217.238,A -85,B 0,C 180,E1 -9360.42,E2 -9360.42} C_VEL
LIN {X 0,Y 545.559,Z 217.276,A -85,B 0,C 180,E1 -9363.783,E2 -9363.783} C_VEL
LIN {X 0,Y 545.568,Z 217.234,A -85,B 0,C 180,E1 -9367.159,E2 -9367.159} C_VEL
LIN {X 0,Y 545.535,Z 217.274,A -85,B 0,C 180,E1 -9370.561,E2 -9370.561} C_VEL
LIN {X 0,Y 545.554,Z 217.276,A -85,B 0,C 180,E1 -9374.001,E2 -9374.001} C_VEL
LIN {X 0,Y 545.566,Z 217.273,A -85,B 0,C 180,E1 -9377.382,E2 -9377.382} C_VEL
LIN {X 0,Y 545.531,Z 217.273,A -85,B 0,C 180,E1 -9380.717,E2 -9380.717} C_VEL
LIN {X 0,Y 545.544,Z 217.269,A -85,B 0,C 180,E1 -9384.125,E2 -9384.125} C_VEL
LIN {X 0,Y 545.569,Z 217.267,A -85,B 0,C 180,E1 -9387.507,E2 -9387.507} C_VEL
LIN {X 0,Y 545.524,Z 217.277,A -85,B 0,C 180,E1 -9390.756,E2 -9390.756} C_VEL
LIN {X 0,Y 545.543,Z 217.269,A -85,B 0,C 180,E1 -9394.115,E2 -9394.115} C_VEL
LIN {X 0,Y 545.572,Z 217.42,A -85,B 0,C 180,E1 -9396.002,E2 -9396.002} C_VEL
LIN {X 0,Y 546.946,Z 220.925,A -85,B 0,C 180,E1 -9396.452,E2 -9396.452} C_VEL
LIN {X 0,Y 548.095,Z 223.012,A -85,B 0,C 180,E1 -9396.754,E2 -9396.754} C_VEL
LIN {X 0,Y 552.553,Z 231.732,A -85,B 0,C 180,E1 -9397.971,E2 -9397.971} C_VEL
LIN {X 0,Y 562.666,Z 251.502,A -85,B 0,C 180,E1 -9400.572,E2 -9400.572} C_VEL
LIN {X 0,Y 575.207,Z 277.134,A -85,B 0,C 180,E1 -9403.639,E2 -9403.639} C_VEL
LIN {X 0,Y 581.285,Z 289.975,A -85,B 0,C 180,E1 -9405.06,E2 -9405.06} C_VEL
LIN {X 0,Y 579.224,Z 311.616,A -85,B 0,C 180,E1 -9406.301,E2 -9406.301} C_VEL
LIN {X 0,Y 582.067,Z 336.568,A -85,B 0,C 180,E1 -9406.945,E2 -9406.945} C_VEL
LIN {X 0,Y 575.098,Z 576.403,A -85,B 0,C 180,E1 -9410.45,E2 -9410.45} C_VEL
LIN {X 0,Y 572.164,Z 692.789,A -85,B 0,C 180,E1 -9412.111,E2 -9412.111} C_VEL
LIN {X 0,Y 570.889,Z 717.376,A -85,B 0,C 180,E1 -9412.632,E2 -9412.632} C_VEL
LIN {X 0,Y 569.353,Z 740.821,A -85,B 0,C 180,E1 -9413.29,E2 -9413.29} C_VEL
LIN {X 0,Y 567.45,Z 764.117,A -85,B 0,C 180,E1 -9414.134,E2 -9414.134} C_VEL
LIN {X 0,Y 565.393,Z 786.321,A -85,B 0,C 180,E1 -9415.103,E2 -9415.103} C_VEL
LIN {X 0,Y 563.033,Z 808.895,A -85,B 0,C 180,E1 -9416.301,E2 -9416.301} C_VEL
LIN {X 0,Y 560.642,Z 830.726,A -85,B 0,C 180,E1 -9417.653,E2 -9417.653} C_VEL
LIN {X 0,Y 558.234,Z 850.811,A -85,B 0,C 180,E1 -9419.119,E2 -9419.119} C_VEL
LIN {X 0,Y 555.877,Z 870.326,A -85,B 0,C 180,E1 -9420.739,E2 -9420.739} C_VEL
LIN {X 0,Y 553.596,Z 888.677,A -85,B 0,C 180,E1 -9422.517,E2 -9422.517} C_VEL
LIN {X 0,Y 551.489,Z 906.198,A -85,B 0,C 180,E1 -9424.437,E2 -9424.437} C_VEL
LIN {X 0,Y 549.661,Z 921.747,A -85,B 0,C 180,E1 -9426.409,E2 -9426.409} C_VEL
LIN {X 0,Y 548.068,Z 936.356,A -85,B 0,C 180,E1 -9428.504,E2 -9428.504} C_VEL
LIN {X 0,Y 546.725,Z 949.932,A -85,B 0,C 180,E1 -9430.78,E2 -9430.78} C_VEL
LIN {X 0,Y 545.711,Z 961.807,A -85,B 0,C 180,E1 -9433.062,E2 -9433.062} C_VEL
LIN {X 0,Y 544.968,Z 972.165,A -85,B 0,C 180,E1 -9435.442,E2 -9435.442} C_VEL
LIN {X 0,Y 544.478,Z 980.864,A -85,B 0,C 180,E1 -9437.808,E2 -9437.808} C_VEL
LIN {X 0,Y 544.195,Z 988.079,A -85,B 0,C 180,E1 -9440.268,E2 -9440.268} C_VEL
LIN {X 0,Y 544.033,Z 992.996,A -85,B 0,C 180,E1 -9442.396,E2 -9442.396} C_VEL
LIN {X 0,Y 543.977,Z 997.187,A -85,B 0,C 180,E1 -9444.833,E2 -9444.833} C_VEL
LIN {X 0,Y 543.972,Z 999.563,A -85,B 0,C 180,E1 -9447.155,E2 -9447.155} C_VEL
LIN {X 0,Y 543.978,Z 1000.543,A -85,B 0,C 180,E1 -9449.263,E2 -9449.263} C_VEL
LIN {X 0,Y 543.995,Z 1000.31,A -85,B 0,C 180,E1 -9451.58,E2 -9451.58} C_VEL
LIN {X 0,Y 544.008,Z 998.31,A -85,B 0,C 180,E1 -9454.111,E2 -9454.111} C_VEL
LIN {X 0,Y 544.031,Z 995.184,A -85,B 0,C 180,E1 -9456.331,E2 -9456.331} C_VEL
LIN {X 0,Y 544.125,Z 989.937,A -85,B 0,C 180,E1 -9458.88,E2 -9458.88} C_VEL
LIN {X 0,Y 544.338,Z 983.75,A -85,B 0,C 180,E1 -9461.121,E2 -9461.121} C_VEL
LIN {X 0,Y 544.735,Z 975.699,A -85,B 0,C 180,E1 -9463.481,E2 -9463.481} C_VEL
LIN {X 0,Y 545.341,Z 965.751,A -85,B 0,C 180,E1 -9465.854,E2 -9465.854} C_VEL
LIN {X 0,Y 546.105,Z 955.604,A -85,B 0,C 180,E1 -9467.915,E2 -9467.915} C_VEL
LIN {X 0,Y 547.279,Z 941.8,A -85,B 0,C 180,E1 -9470.312,E2 -9470.312} C_VEL
LIN {X 0,Y 548.498,Z 928.642,A -85,B 0,C 180,E1 -9472.283,E2 -9472.283} C_VEL
LIN {X 0,Y 550.212,Z 911.802,A -85,B 0,C 180,E1 -9474.478,E2 -9474.478} C_VEL
LIN {X 0,Y 551.836,Z 896.243,A -85,B 0,C 180,E1 -9476.245,E2 -9476.245} C_VEL
LIN {X 0,Y 553.947,Z 876.817,A -85,B 0,C 180,E1 -9478.177,E2 -9478.177} C_VEL
LIN {X 0,Y 555.851,Z 859.161,A -85,B 0,C 180,E1 -9479.708,E2 -9479.708} C_VEL
LIN {X 0,Y 558.218,Z 836.465,A -85,B 0,C 180,E1 -9481.416,E2 -9481.416} C_VEL
LIN {X 0,Y 560.236,Z 816.516,A -85,B 0,C 180,E1 -9482.707,E2 -9482.707} C_VEL
LIN {X 0,Y 562.292,Z 794.189,A -85,B 0,C 180,E1 -9483.943,E2 -9483.943} C_VEL
LIN {X 0,Y 564.081,Z 773.206,A -85,B 0,C 180,E1 -9484.928,E2 -9484.928} C_VEL
LIN {X 0,Y 565.884,Z 749.209,A -85,B 0,C 180,E1 -9485.856,E2 -9485.856} C_VEL
LIN {X 0,Y 567.361,Z 726.472,A -85,B 0,C 180,E1 -9486.561,E2 -9486.561} C_VEL
LIN {X 0,Y 568.594,Z 702.091,A -85,B 0,C 180,E1 -9487.129,E2 -9487.129} C_VEL
LIN {X 0,Y 569.338,Z 679.341,A -85,B 0,C 180,E1 -9487.512,E2 -9487.512} C_VEL
LIN {X 0,Y 571.757,Z 561.36,A -85,B 0,C 180,E1 -9489.146,E2 -9489.146} C_VEL
LIN {X 0,Y 574.925,Z 458.823,A -85,B 0,C 180,E1 -9490.727,E2 -9490.727} C_VEL
LIN {X 0,Y 579.149,Z 367.753,A -85,B 0,C 180,E1 -9492.266,E2 -9492.266} C_VEL
LIN {X 0,Y 581.054,Z 335.093,A -85,B 0,C 180,E1 -9492.855,E2 -9492.855} C_VEL
LIN {X 0,Y 587.23,Z 314.419,A -85,B 0,C 180,E1 -9494.484,E2 -9494.484} C_VEL
LIN {X 0,Y 592.696,Z 300.447,A -85,B 0,C 180,E1 -9495.699,E2 -9495.699} C_VEL
LIN {X 0,Y 592.266,Z 297.133,A -85,B 0,C 180,E1 -9496.863,E2 -9496.863} C_VEL
LIN {X 0,Y 592.264,Z 295.324,A -85,B 0,C 180,E1 -9498.175,E2 -9498.175} C_VEL
LIN {X 0,Y 591.776,Z 297.266,A -85,B 0,C 180,E1 -9499.674,E2 -9499.674} C_VEL
LIN {X 0,Y 591.615,Z 299.404,A -85,B 0,C 180,E1 -9500.419,E2 -9500.419} C_VEL
LIN {X 0,Y 584.152,Z 317.161,A -85,B 0,C 180,E1 -9502.208,E2 -9502.208} C_VEL
LIN {X 0,Y 576.831,Z 341.117,A -85,B 0,C 180,E1 -9504.439,E2 -9504.439} C_VEL
LIN {X 0,Y 570.306,Z 371.749,A -85,B 0,C 180,E1 -9507.077,E2 -9507.077} C_VEL
LIN {X 0,Y 564.785,Z 407.956,A -85,B 0,C 180,E1 -9509.974,E2 -9509.974} C_VEL
LIN {X 0,Y 567.185,Z 438.405,A -85,B 0,C 180,E1 -9511.397,E2 -9511.397} C_VEL
LIN {X 0,Y 569.308,Z 473.337,A -85,B 0,C 180,E1 -9512.783,E2 -9512.783} C_VEL
LIN {X 0,Y 570.357,Z 498.769,A -85,B 0,C 180,E1 -9513.657,E2 -9513.657} C_VEL
LIN {X 0,Y 562.703,Z 603.388,A -85,B 0,C 180,E1 -9515.926,E2 -9515.926} C_VEL
LIN {X 0,Y 557.941,Z 688.582,A -85,B 0,C 180,E1 -9517.737,E2 -9517.737} C_VEL
LIN {X 0,Y 556.623,Z 711.497,A -85,B 0,C 180,E1 -9518.417,E2 -9518.417} C_VEL
LIN {X 0,Y 555.349,Z 732.232,A -85,B 0,C 180,E1 -9519.225,E2 -9519.225} C_VEL
LIN {X 0,Y 554.022,Z 752.678,A -85,B 0,C 180,E1 -9520.221,E2 -9520.221} C_VEL
LIN {X 0,Y 552.772,Z 771.115,A -85,B 0,C 180,E1 -9521.327,E2 -9521.327} C_VEL
LIN {X 0,Y 551.484,Z 789.197,A -85,B 0,C 180,E1 -9522.647,E2 -9522.647} C_VEL
LIN {X 0,Y 550.312,Z 804.791,A -85,B 0,C 180,E1 -9524.022,E2 -9524.022} C_VEL
LIN {X 0,Y 549.264,Z 818.297,A -85,B 0,C 180,E1 -9525.45,E2 -9525.45} C_VEL
LIN {X 0,Y 548.289,Z 830.809,A -85,B 0,C 180,E1 -9527.038,E2 -9527.038} C_VEL
LIN {X 0,Y 547.421,Z 841.703,A -85,B 0,C 180,E1 -9528.729,E2 -9528.729} C_VEL
LIN {X 0,Y 546.686,Z 850.984,A -85,B 0,C 180,E1 -9530.525,E2 -9530.525} C_VEL
LIN {X 0,Y 546.133,Z 858.24,A -85,B 0,C 180,E1 -9532.319,E2 -9532.319} C_VEL
LIN {X 0,Y 545.712,Z 863.903,A -85,B 0,C 180,E1 -9534.216,E2 -9534.216} C_VEL
LIN {X 0,Y 545.397,Z 867.699,A -85,B 0,C 180,E1 -9536.11,E2 -9536.11} C_VEL
LIN {X 0,Y 545.189,Z 869.735,A -85,B 0,C 180,E1 -9538.003,E2 -9538.003} C_VEL
LIN {X 0,Y 545.062,Z 870.008,A -85,B 0,C 180,E1 -9540,E2 -9540} C_VEL
LIN {X 0,Y 544.997,Z 868.394,A -85,B 0,C 180,E1 -9541.998,E2 -9541.998} C_VEL
LIN {X 0,Y 545.022,Z 865.153,A -85,B 0,C 180,E1 -9543.892,E2 -9543.892} C_VEL
LIN {X 0,Y 545.145,Z 860.169,A -85,B 0,C 180,E1 -9545.79,E2 -9545.79} C_VEL
LIN {X 0,Y 545.37,Z 853.329,A -85,B 0,C 180,E1 -9547.692,E2 -9547.692} C_VEL
LIN {X 0,Y 545.733,Z 845.011,A -85,B 0,C 180,E1 -9549.491,E2 -9549.491} C_VEL
LIN {X 0,Y 546.275,Z 834.634,A -85,B 0,C 180,E1 -9551.294,E2 -9551.294} C_VEL
LIN {X 0,Y 546.971,Z 822.697,A -85,B 0,C 180,E1 -9552.994,E2 -9552.994} C_VEL
LIN {X 0,Y 547.817,Z 809.197,A -85,B 0,C 180,E1 -9554.589,E2 -9554.589} C_VEL
LIN {X 0,Y 548.794,Z 794.082,A -85,B 0,C 180,E1 -9556.078,E2 -9556.078} C_VEL
LIN {X 0,Y 549.884,Z 777.199,A -85,B 0,C 180,E1 -9557.46,E2 -9557.46} C_VEL
LIN {X 0,Y 550.942,Z 759.953,A -85,B 0,C 180,E1 -9558.628,E2 -9558.628} C_VEL
LIN {X 0,Y 552.012,Z 741.997,A -85,B 0,C 180,E1 -9559.626,E2 -9559.626} C_VEL
LIN {X 0,Y 553.037,Z 722.914,A -85,B 0,C 180,E1 -9560.478,E2 -9560.478} C_VEL
LIN {X 0,Y 553.969,Z 702.7,A -85,B 0,C 180,E1 -9561.175,E2 -9561.175} C_VEL
LIN {X 0,Y 554.788,Z 681.509,A -85,B 0,C 180,E1 -9561.697,E2 -9561.697} C_VEL
LIN {X 0,Y 559.864,Z 492.751,A -85,B 0,C 180,E1 -9564.763,E2 -9564.763} C_VEL
LIN {X 0,Y 555.561,Z 452.559,A -85,B 0,C 180,E1 -9565.706,E2 -9565.706} C_VEL
LIN {X 0,Y 558.757,Z 398.884,A -85,B 0,C 180,E1 -9569.303,E2 -9569.303} C_VEL
LIN {X 0,Y 562.093,Z 348.261,A -85,B 0,C 180,E1 -9572.737,E2 -9572.737} C_VEL
LIN {X 0,Y 565.901,Z 296.072,A -85,B 0,C 180,E1 -9576.321,E2 -9576.321} C_VEL
LIN {X 0,Y 567.638,Z 273.459,A -85,B 0,C 180,E1 -9577.894,E2 -9577.894} C_VEL
LIN {X 0,Y 559.201,Z 250.997,A -85,B 0,C 180,E1 -9580.226,E2 -9580.226} C_VEL
LIN {X 0,Y 549.663,Z 227.521,A -85,B 0,C 180,E1 -9582.853,E2 -9582.853} C_VEL
LIN {X 0,Y 545.622,Z 217.809,A -85,B 0,C 180,E1 -9584.009,E2 -9584.009} C_VEL
LIN {X 0,Y 546.762,Z 220.631,A -85,B 0,C 180,E1 -9584.314,E2 -9584.314} C_VEL
LIN {X 0,Y 547.967,Z 222.455,A -85,B 0,C 180,E1 -9584.556,E2 -9584.556} C_VEL
LIN {X 0,Y 556.854,Z 240.409,A -85,B 0,C 180,E1 -9586.654,E2 -9586.654} C_VEL
LIN {X 0,Y 557.809,Z 242.388,A -85,B 0,C 180,E1 -9586.882,E2 -9586.882} C_VEL
LIN {X 0,Y 559.194,Z 248.018,A -85,B 0,C 180,E1 -9587.413,E2 -9587.413} C_VEL
LIN {X 0,Y 560.151,Z 264.918,A -85,B 0,C 180,E1 -9588.731,E2 -9588.731} C_VEL
LIN {X 0,Y 561.338,Z 269.652,A -85,B 0,C 180,E1 -9589.197,E2 -9589.197} C_VEL
LIN {X 0,Y 567.742,Z 287.266,A -85,B 0,C 180,E1 -9591.118,E2 -9591.118} C_VEL
LIN {X 0,Y 567.028,Z 328.039,A -85,B 0,C 180,E1 -9593.978,E2 -9593.978} C_VEL
LIN {X 0,Y 567.18,Z 345.277,A -85,B 0,C 180,E1 -9595.099,E2 -9595.099} C_VEL
LIN {X 0,Y 565.296,Z 354.489,A -85,B 0,C 180,E1 -9595.445,E2 -9595.445} C_VEL
LIN {X 0,Y 562.822,Z 445.712,A -85,B 0,C 180,E1 -9596.748,E2 -9596.748} C_VEL
LIN {X 0,Y 559.596,Z 528.217,A -85,B 0,C 180,E1 -9598.114,E2 -9598.114} C_VEL
LIN {X 0,Y 555.257,Z 623.232,A -85,B 0,C 180,E1 -9599.903,E2 -9599.903} C_VEL
LIN {X 0,Y 554.368,Z 646.878,A -85,B 0,C 180,E1 -9600.472,E2 -9600.472} C_VEL
LIN {X 0,Y 553.181,Z 669.205,A -85,B 0,C 180,E1 -9601.203,E2 -9601.203} C_VEL
LIN {X 0,Y 551.745,Z 690.945,A -85,B 0,C 180,E1 -9602.124,E2 -9602.124} C_VEL
LIN {X 0,Y 550.167,Z 710.976,A -85,B 0,C 180,E1 -9603.172,E2 -9603.172} C_VEL
LIN {X 0,Y 548.428,Z 730.474,A -85,B 0,C 180,E1 -9604.399,E2 -9604.399} C_VEL
LIN {X 0,Y 546.525,Z 749.886,A -85,B 0,C 180,E1 -9605.864,E2 -9605.864} C_VEL
LIN {X 0,Y 544.687,Z 767.505,A -85,B 0,C 180,E1 -9607.439,E2 -9607.439} C_VEL
LIN {X 0,Y 542.971,Z 783.58,A -85,B 0,C 180,E1 -9609.125,E2 -9609.125} C_VEL
LIN {X 0,Y 541.341,Z 799.064,A -85,B 0,C 180,E1 -9611.029,E2 -9611.029} C_VEL
LIN {X 0,Y 539.973,Z 812.571,A -85,B 0,C 180,E1 -9612.988,E2 -9612.988} C_VEL
LIN {X 0,Y 538.893,Z 824.057,A -85,B 0,C 180,E1 -9614.944,E2 -9614.944} C_VEL
LIN {X 0,Y 537.996,Z 834.666,A -85,B 0,C 180,E1 -9617.113,E2 -9617.113} C_VEL
LIN {X 0,Y 537.366,Z 843.29,A -85,B 0,C 180,E1 -9619.276,E2 -9619.276} C_VEL
LIN {X 0,Y 536.938,Z 850.477,A -85,B 0,C 180,E1 -9621.54,E2 -9621.54} C_VEL
LIN {X 0,Y 536.699,Z 855.899,A -85,B 0,C 180,E1 -9623.797,E2 -9623.797} C_VEL
LIN {X 0,Y 536.578,Z 859.644,A -85,B 0,C 180,E1 -9626.046,E2 -9626.046} C_VEL
LIN {X 0,Y 536.52,Z 861.661,A -85,B 0,C 180,E1 -9628.291,E2 -9628.291} C_VEL
LIN {X 0,Y 536.5,Z 862.115,A -85,B 0,C 180,E1 -9630.534,E2 -9630.534} C_VEL
LIN {X 0,Y 536.535,Z 861.09,A -85,B 0,C 180,E1 -9632.689,E2 -9632.689} C_VEL
LIN {X 0,Y 536.616,Z 858.351,A -85,B 0,C 180,E1 -9634.917,E2 -9634.917} C_VEL
LIN {X 0,Y 536.76,Z 853.991,A -85,B 0,C 180,E1 -9637.17,E2 -9637.17} C_VEL
LIN {X 0,Y 537.06,Z 848.228,A -85,B 0,C 180,E1 -9639.337,E2 -9639.337} C_VEL
LIN {X 0,Y 537.582,Z 840.447,A -85,B 0,C 180,E1 -9641.588,E2 -9641.588} C_VEL
LIN {X 0,Y 538.282,Z 831.066,A -85,B 0,C 180,E1 -9643.755,E2 -9643.755} C_VEL
LIN {X 0,Y 539.238,Z 820.299,A -85,B 0,C 180,E1 -9645.818,E2 -9645.818} C_VEL
LIN {X 0,Y 540.484,Z 807.46,A -85,B 0,C 180,E1 -9647.884,E2 -9647.884} C_VEL
LIN {X 0,Y 541.931,Z 793.541,A -85,B 0,C 180,E1 -9649.783,E2 -9649.783} C_VEL
LIN {X 0,Y 543.588,Z 778.05,A -85,B 0,C 180,E1 -9651.585,E2 -9651.585} C_VEL
LIN {X 0,Y 545.433,Z 760.64,A -85,B 0,C 180,E1 -9653.301,E2 -9653.301} C_VEL
LIN {X 0,Y 547.234,Z 742.771,A -85,B 0,C 180,E1 -9654.793,E2 -9654.793} C_VEL
LIN {X 0,Y 549.001,Z 724.32,A -85,B 0,C 180,E1 -9656.1,E2 -9656.1} C_VEL
LIN {X 0,Y 550.7,Z 704.388,A -85,B 0,C 180,E1 -9657.288,E2 -9657.288} C_VEL
LIN {X 0,Y 552.219,Z 684.621,A -85,B 0,C 180,E1 -9658.261,E2 -9658.261} C_VEL
LIN {X 0,Y 553.591,Z 663.149,A -85,B 0,C 180,E1 -9659.114,E2 -9659.114} C_VEL
LIN {X 0,Y 554.663,Z 640.615,A -85,B 0,C 180,E1 -9659.797,E2 -9659.797} C_VEL
LIN {X 0,Y 556.053,Z 605.062,A -85,B 0,C 180,E1 -9660.551,E2 -9660.551} C_VEL
LIN {X 0,Y 560.307,Z 512.148,A -85,B 0,C 180,E1 -9662.259,E2 -9662.259} C_VEL
LIN {X 0,Y 563.191,Z 435.44,A -85,B 0,C 180,E1 -9663.501,E2 -9663.501} C_VEL
LIN {X 0,Y 565.436,Z 353.224,A -85,B 0,C 180,E1 -9664.678,E2 -9664.678} C_VEL
LIN {X 0,Y 567.211,Z 344.978,A -85,B 0,C 180,E1 -9665.015,E2 -9665.015} C_VEL
LIN {X 0,Y 567.263,Z 309.602,A -85,B 0,C 180,E1 -9667.383,E2 -9667.383} C_VEL
LIN {X 0,Y 567.719,Z 286.667,A -85,B 0,C 180,E1 -9669.04,E2 -9669.04} C_VEL
LIN {X 0,Y 559.678,Z 265.46,A -85,B 0,C 180,E1 -9671.379,E2 -9671.379} C_VEL
LIN {X 0,Y 551.645,Z 246.659,A -85,B 0,C 180,E1 -9673.533,E2 -9673.533} C_VEL
LIN {X 0,Y 543.96,Z 231.051,A -85,B 0,C 180,E1 -9675.397,E2 -9675.397} C_VEL
LIN {X 0,Y 539.479,Z 222.458,A -85,B 0,C 180,E1 -9676.443,E2 -9676.443} C_VEL
LIN {X 0,Y 537.813,Z 219.316,A -85,B 0,C 180,E1 -9676.829,E2 -9676.829} C_VEL
LIN {X 0,Y 537.603,Z 218.255,A -85,B 0,C 180,E1 -9676.954,E2 -9676.954} C_VEL
LIN {X 0,Y 537.624,Z 218.253,A -85,B 0,C 180,E1 -9680.351,E2 -9680.351} C_VEL
LIN {X 0,Y 537.621,Z 218.247,A -85,B 0,C 180,E1 -9683.821,E2 -9683.821} C_VEL
LIN {X 0,Y 537.606,Z 218.241,A -85,B 0,C 180,E1 -9687.232,E2 -9687.232} C_VEL
LIN {X 0,Y 537.626,Z 218.247,A -85,B 0,C 180,E1 -9690.594,E2 -9690.594} C_VEL
LIN {X 0,Y 537.617,Z 218.262,A -85,B 0,C 180,E1 -9694.083,E2 -9694.083} C_VEL
LIN {X 0,Y 537.612,Z 218.238,A -85,B 0,C 180,E1 -9697.472,E2 -9697.472} C_VEL
LIN {X 0,Y 537.62,Z 218.24,A -85,B 0,C 180,E1 -9700.893,E2 -9700.893} C_VEL
LIN {X 0,Y 537.61,Z 218.26,A -85,B 0,C 180,E1 -9704.355,E2 -9704.355} C_VEL
LIN {X 0,Y 537.616,Z 218.228,A -85,B 0,C 180,E1 -9707.759,E2 -9707.759} C_VEL
LIN {X 0,Y 537.619,Z 218.261,A -85,B 0,C 180,E1 -9711.228,E2 -9711.228} C_VEL
LIN {X 0,Y 537.604,Z 218.231,A -85,B 0,C 180,E1 -9714.557,E2 -9714.557} C_VEL
LIN {X 0,Y 537.614,Z 218.259,A -85,B 0,C 180,E1 -9717.975,E2 -9717.975} C_VEL
LIN {X 0,Y 537.618,Z 218.229,A -85,B 0,C 180,E1 -9721.385,E2 -9721.385} C_VEL
LIN {X 0,Y 537.609,Z 218.258,A -85,B 0,C 180,E1 -9724.801,E2 -9724.801} C_VEL
LIN {X 0,Y 537.597,Z 218.237,A -85,B 0,C 180,E1 -9728.234,E2 -9728.234} C_VEL
LIN {X 0,Y 537.624,Z 218.262,A -85,B 0,C 180,E1 -9731.587,E2 -9731.587} C_VEL
LIN {X 0,Y 537.609,Z 218.258,A -85,B 0,C 180,E1 -9734.983,E2 -9734.983} C_VEL
LIN {X 0,Y 537.592,Z 218.257,A -85,B 0,C 180,E1 -9738.433,E2 -9738.433} C_VEL
LIN {X 0,Y 537.627,Z 218.256,A -85,B 0,C 180,E1 -9741.867,E2 -9741.867} C_VEL
LIN {X 0,Y 537.623,Z 218.261,A -85,B 0,C 180,E1 -9745.327,E2 -9745.327} C_VEL
LIN {X 0,Y 537.588,Z 218.263,A -85,B 0,C 180,E1 -9748.677,E2 -9748.677} C_VEL
LIN {X 0,Y 537.612,Z 218.258,A -85,B 0,C 180,E1 -9752.01,E2 -9752.01} C_VEL
LIN {X 0,Y 537.608,Z 218.319,A -85,B 0,C 180,E1 -9755.144,E2 -9755.144} C_VEL
LIN {X 0,Y 539.036,Z 221.888,A -85,B 0,C 180,E1 -9755.624,E2 -9755.624} C_VEL
LIN {X 0,Y 540.145,Z 223.959,A -85,B 0,C 180,E1 -9755.932,E2 -9755.932} C_VEL
LIN {X 0,Y 547.148,Z 237.722,A -85,B 0,C 180,E1 -9757.865,E2 -9757.865} C_VEL
LIN {X 0,Y 555.793,Z 254.685,A -85,B 0,C 180,E1 -9760.13,E2 -9760.13} C_VEL
LIN {X 0,Y 567.777,Z 279.06,A -85,B 0,C 180,E1 -9763.102,E2 -9763.102} C_VEL
LIN {X 0,Y 574.624,Z 293.591,A -85,B 0,C 180,E1 -9764.734,E2 -9764.734} C_VEL
LIN {X 0,Y 572.789,Z 312.388,A -85,B 0,C 180,E1 -9765.819,E2 -9765.819} C_VEL
LIN {X 0,Y 575.609,Z 337.913,A -85,B 0,C 180,E1 -9766.489,E2 -9766.489} C_VEL
LIN {X 0,Y 568.399,Z 574.17,A -85,B 0,C 180,E1 -9769.987,E2 -9769.987} C_VEL
LIN {X 0,Y 565.24,Z 692.907,A -85,B 0,C 180,E1 -9771.707,E2 -9771.707} C_VEL
LIN {X 0,Y 563.911,Z 717.312,A -85,B 0,C 180,E1 -9772.231,E2 -9772.231} C_VEL
LIN {X 0,Y 562.316,Z 740.745,A -85,B 0,C 180,E1 -9772.898,E2 -9772.898} C_VEL
LIN {X 0,Y 560.358,Z 763.761,A -85,B 0,C 180,E1 -9773.741,E2 -9773.741} C_VEL
LIN {X 0,Y 558.236,Z 785.814,A -85,B 0,C 180,E1 -9774.715,E2 -9774.715} C_VEL
LIN {X 0,Y 555.841,Z 808.023,A -85,B 0,C 180,E1 -9775.899,E2 -9775.899} C_VEL
LIN {X 0,Y 553.354,Z 829.831,A -85,B 0,C 180,E1 -9777.256,E2 -9777.256} C_VEL
LIN {X 0,Y 550.83,Z 850.208,A -85,B 0,C 180,E1 -9778.758,E2 -9778.758} C_VEL
LIN {X 0,Y 548.389,Z 869.628,A -85,B 0,C 180,E1 -9780.388,E2 -9780.388} C_VEL
LIN {X 0,Y 545.99,Z 888.123,A -85,B 0,C 180,E1 -9782.195,E2 -9782.195} C_VEL
LIN {X 0,Y 543.894,Z 904.929,A -85,B 0,C 180,E1 -9784.053,E2 -9784.053} C_VEL
LIN {X 0,Y 541.864,Z 921.378,A -85,B 0,C 180,E1 -9786.164,E2 -9786.164} C_VEL
LIN {X 0,Y 540.205,Z 936.094,A -85,B 0,C 180,E1 -9788.307,E2 -9788.307} C_VEL
LIN {X 0,Y 538.814,Z 949.512,A -85,B 0,C 180,E1 -9790.599,E2 -9790.599} C_VEL
LIN {X 0,Y 537.763,Z 961.35,A -85,B 0,C 180,E1 -9792.916,E2 -9792.916} C_VEL
LIN {X 0,Y 536.997,Z 971.653,A -85,B 0,C 180,E1 -9795.331,E2 -9795.331} C_VEL
LIN {X 0,Y 536.496,Z 980.32,A -85,B 0,C 180,E1 -9797.733,E2 -9797.733} C_VEL
LIN {X 0,Y 536.213,Z 987.47,A -85,B 0,C 180,E1 -9800.23,E2 -9800.23} C_VEL
LIN {X 0,Y 536.056,Z 992.559,A -85,B 0,C 180,E1 -9802.498,E2 -9802.498} C_VEL
LIN {X 0,Y 536.021,Z 996.702,A -85,B 0,C 180,E1 -9805.078,E2 -9805.078} C_VEL
LIN {X 0,Y 536.018,Z 998.855,A -85,B 0,C 180,E1 -9807.327,E2 -9807.327} C_VEL
LIN {X 0,Y 536.024,Z 999.722,A -85,B 0,C 180,E1 -9809.466,E2 -9809.466} C_VEL
LIN {X 0,Y 536.049,Z 999.206,A -85,B 0,C 180,E1 -9812.031,E2 -9812.031} C_VEL
LIN {X 0,Y 536.052,Z 997.162,A -85,B 0,C 180,E1 -9814.386,E2 -9814.386} C_VEL
LIN {X 0,Y 536.086,Z 993.523,A -85,B 0,C 180,E1 -9816.856,E2 -9816.856} C_VEL
LIN {X 0,Y 536.215,Z 987.846,A -85,B 0,C 180,E1 -9819.446,E2 -9819.446} C_VEL
LIN {X 0,Y 536.436,Z 981.355,A -85,B 0,C 180,E1 -9821.723,E2 -9821.723} C_VEL
LIN {X 0,Y 536.902,Z 972.446,A -85,B 0,C 180,E1 -9824.231,E2 -9824.231} C_VEL
LIN {X 0,Y 537.486,Z 963.529,A -85,B 0,C 180,E1 -9826.314,E2 -9826.314} C_VEL
LIN {X 0,Y 538.381,Z 952.034,A -85,B 0,C 180,E1 -9828.629,E2 -9828.629} C_VEL
LIN {X 0,Y 539.558,Z 938.995,A -85,B 0,C 180,E1 -9830.843,E2 -9830.843} C_VEL
LIN {X 0,Y 541.046,Z 924.362,A -85,B 0,C 180,E1 -9833.024,E2 -9833.024} C_VEL
LIN {X 0,Y 542.72,Z 908.339,A -85,B 0,C 180,E1 -9835.071,E2 -9835.071} C_VEL
LIN {X 0,Y 544.653,Z 891.221,A -85,B 0,C 180,E1 -9837.003,E2 -9837.003} C_VEL
LIN {X 0,Y 546.634,Z 873.266,A -85,B 0,C 180,E1 -9838.756,E2 -9838.756} C_VEL
LIN {X 0,Y 548.843,Z 853.871,A -85,B 0,C 180,E1 -9840.429,E2 -9840.429} C_VEL
LIN {X 0,Y 551.07,Z 833.524,A -85,B 0,C 180,E1 -9841.932,E2 -9841.932} C_VEL
LIN {X 0,Y 553.329,Z 811.96,A -85,B 0,C 180,E1 -9843.322,E2 -9843.322} C_VEL
LIN {X 0,Y 555.351,Z 790.52,A -85,B 0,C 180,E1 -9844.489,E2 -9844.489} C_VEL
LIN {X 0,Y 557.466,Z 767.194,A -85,B 0,C 180,E1 -9845.562,E2 -9845.562} C_VEL
LIN {X 0,Y 559.208,Z 744.36,A -85,B 0,C 180,E1 -9846.415,E2 -9846.415} C_VEL
LIN {X 0,Y 560.836,Z 719.263,A -85,B 0,C 180,E1 -9847.156,E2 -9847.156} C_VEL
LIN {X 0,Y 561.925,Z 697.13,A -85,B 0,C 180,E1 -9847.647,E2 -9847.647} C_VEL
LIN {X 0,Y 562.89,Z 662.167,A -85,B 0,C 180,E1 -9848.177,E2 -9848.177} C_VEL
LIN {X 0,Y 565.438,Z 555.973,A -85,B 0,C 180,E1 -9849.702,E2 -9849.702} C_VEL
LIN {X 0,Y 568.875,Z 459.993,A -85,B 0,C 180,E1 -9851.242,E2 -9851.242} C_VEL
LIN {X 0,Y 573.522,Z 371.719,A -85,B 0,C 180,E1 -9852.787,E2 -9852.787} C_VEL
LIN {X 0,Y 575.928,Z 337.583,A -85,B 0,C 180,E1 -9853.433,E2 -9853.433} C_VEL
LIN {X 0,Y 582.392,Z 318.422,A -85,B 0,C 180,E1 -9854.98,E2 -9854.98} C_VEL
LIN {X 0,Y 587.759,Z 305.833,A -85,B 0,C 180,E1 -9856.092,E2 -9856.092} C_VEL
LIN {X 0,Y 587.512,Z 303.318,A -85,B 0,C 180,E1 -9857.096,E2 -9857.096} C_VEL
LIN {X 0,Y 587.613,Z 301.92,A -85,B 0,C 180,E1 -9858.186,E2 -9858.186} C_VEL
LIN {X 0,Y 587.057,Z 303.686,A -85,B 0,C 180,E1 -9859.583,E2 -9859.583} C_VEL
LIN {X 0,Y 586.853,Z 304.967,A -85,B 0,C 180,E1 -9860.033,E2 -9860.033} C_VEL
LIN {X 0,Y 578.996,Z 322.192,A -85,B 0,C 180,E1 -9861.812,E2 -9861.812} C_VEL
LIN {X 0,Y 571.699,Z 343.811,A -85,B 0,C 180,E1 -9863.885,E2 -9863.885} C_VEL
LIN {X 0,Y 564.744,Z 372.896,A -85,B 0,C 180,E1 -9866.468,E2 -9866.468} C_VEL
LIN {X 0,Y 559.333,Z 404.006,A -85,B 0,C 180,E1 -9869.035,E2 -9869.035} C_VEL
LIN {X 0,Y 561.123,Z 431.011,A -85,B 0,C 180,E1 -9870.396,E2 -9870.396} C_VEL
LIN {X 0,Y 562.74,Z 458.292,A -85,B 0,C 180,E1 -9871.586,E2 -9871.586} C_VEL
LIN {X 0,Y 564.237,Z 492.411,A -85,B 0,C 180,E1 -9872.885,E2 -9872.885} C_VEL
LIN {X 0,Y 564.296,Z 500.86,A -85,B 0,C 180,E1 -9873.152,E2 -9873.152} C_VEL
LIN {X 0,Y 555.896,Z 607.992,A -85,B 0,C 180,E1 -9875.545,E2 -9875.545} C_VEL
LIN {X 0,Y 550.995,Z 689.896,A -85,B 0,C 180,E1 -9877.342,E2 -9877.342} C_VEL
LIN {X 0,Y 549.559,Z 712.618,A -85,B 0,C 180,E1 -9878.044,E2 -9878.044} C_VEL
LIN {X 0,Y 548.102,Z 734.86,A -85,B 0,C 180,E1 -9878.938,E2 -9878.938} C_VEL
LIN {X 0,Y 546.7,Z 754.813,A -85,B 0,C 180,E1 -9879.944,E2 -9879.944} C_VEL
LIN {X 0,Y 545.257,Z 774.457,A -85,B 0,C 180,E1 -9881.171,E2 -9881.171} C_VEL
LIN {X 0,Y 544.007,Z 790.835,A -85,B 0,C 180,E1 -9882.402,E2 -9882.402} C_VEL
LIN {X 0,Y 542.76,Z 806.281,A -85,B 0,C 180,E1 -9883.794,E2 -9883.794} C_VEL
LIN {X 0,Y 541.656,Z 819.766,A -85,B 0,C 180,E1 -9885.241,E2 -9885.241} C_VEL
LIN {X 0,Y 540.606,Z 832.173,A -85,B 0,C 180,E1 -9886.85,E2 -9886.85} C_VEL
LIN {X 0,Y 539.697,Z 842.932,A -85,B 0,C 180,E1 -9888.543,E2 -9888.543} C_VEL
LIN {X 0,Y 538.942,Z 851.839,A -85,B 0,C 180,E1 -9890.28,E2 -9890.28} C_VEL
LIN {X 0,Y 538.33,Z 859.145,A -85,B 0,C 180,E1 -9892.1,E2 -9892.1} C_VEL
LIN {X 0,Y 537.866,Z 864.892,A -85,B 0,C 180,E1 -9894.024,E2 -9894.024} C_VEL
LIN {X 0,Y 537.517,Z 868.74,A -85,B 0,C 180,E1 -9895.947,E2 -9895.947} C_VEL
LIN {X 0,Y 537.273,Z 870.862,A -85,B 0,C 180,E1 -9897.974,E2 -9897.974} C_VEL
LIN {X 0,Y 537.137,Z 871.108,A -85,B 0,C 180,E1 -9899.893,E2 -9899.893} C_VEL
LIN {X 0,Y 537.062,Z 869.527,A -85,B 0,C 180,E1 -9901.92,E2 -9901.92} C_VEL
LIN {X 0,Y 537.085,Z 866.053,A -85,B 0,C 180,E1 -9903.95,E2 -9903.95} C_VEL
LIN {X 0,Y 537.214,Z 860.974,A -85,B 0,C 180,E1 -9905.876,E2 -9905.876} C_VEL
LIN {X 0,Y 537.453,Z 854.029,A -85,B 0,C 180,E1 -9907.806,E2 -9907.806} C_VEL
LIN {X 0,Y 537.835,Z 845.598,A -85,B 0,C 180,E1 -9909.632,E2 -9909.632} C_VEL
LIN {X 0,Y 538.407,Z 835.101,A -85,B 0,C 180,E1 -9911.462,E2 -9911.462} C_VEL
LIN {X 0,Y 539.138,Z 823.039,A -85,B 0,C 180,E1 -9913.186,E2 -9913.186} C_VEL
LIN {X 0,Y 540.025,Z 809.408,A -85,B 0,C 180,E1 -9914.804,E2 -9914.804} C_VEL
LIN {X 0,Y 541.048,Z 794.154,A -85,B 0,C 180,E1 -9916.314,E2 -9916.314} C_VEL
LIN {X 0,Y 542.144,Z 777.833,A -85,B 0,C 180,E1 -9917.662,E2 -9917.662} C_VEL
LIN {X 0,Y 543.242,Z 760.571,A -85,B 0,C 180,E1 -9918.846,E2 -9918.846} C_VEL
LIN {X 0,Y 544.376,Z 742.252,A -85,B 0,C 180,E1 -9919.877,E2 -9919.877} C_VEL
LIN {X 0,Y 545.486,Z 722.321,A -85,B 0,C 180,E1 -9920.775,E2 -9920.775} C_VEL
LIN {X 0,Y 546.474,Z 701.565,A -85,B 0,C 180,E1 -9921.49,E2 -9921.49} C_VEL
LIN {X 0,Y 547.309,Z 680.19,A -85,B 0,C 180,E1 -9922.009,E2 -9922.009} C_VEL
LIN {X 0,Y 552.595,Z 493.47,A -85,B 0,C 180,E1 -9925.107,E2 -9925.107} C_VEL
LIN {X 0,Y 548.2,Z 451.265,A -85,B 0,C 180,E1 -9926.135,E2 -9926.135} C_VEL
LIN {X 0,Y 551.51,Z 398.377,A -85,B 0,C 180,E1 -9929.723,E2 -9929.723} C_VEL
LIN {X 0,Y 554.973,Z 348.44,A -85,B 0,C 180,E1 -9933.149,E2 -9933.149} C_VEL
LIN {X 0,Y 558.933,Z 296.84,A -85,B 0,C 180,E1 -9936.732,E2 -9936.732} C_VEL
LIN {X 0,Y 560.457,Z 276.111,A -85,B 0,C 180,E1 -9938.198,E2 -9938.198} C_VEL
LIN {X 0,Y 552.254,Z 254.309,A -85,B 0,C 180,E1 -9940.497,E2 -9940.497} C_VEL
LIN {X 0,Y 543.152,Z 231.849,A -85,B 0,C 180,E1 -9943.043,E2 -9943.043} C_VEL
LIN {X 0,Y 540.134,Z 224.771,A -85,B 0,C 180,E1 -9943.89,E2 -9943.89} C_VEL
LIN {X 0,Y 542.145,Z 227.323,A -85,B 0,C 180,E1 -9944.273,E2 -9944.273} C_VEL
LIN {X 0,Y 551.923,Z 247.289,A -85,B 0,C 180,E1 -9946.644,E2 -9946.644} C_VEL
LIN {X 0,Y 560.18,Z 266.792,A -85,B 0,C 180,E1 -9948.873,E2 -9948.873} C_VEL
LIN {X 0,Y 561.338,Z 269.652,A -85,B 0,C 180,E1 -9949.197,E2 -9949.197} C_VEL
LIN {X 0,Y 562.612,Z 275.26,A -85,B 0,C 180,E1 -9949.731,E2 -9949.731} C_VEL
LIN {X 0,Y 562.528,Z 283.43,A -85,B 0,C 180,E1 -9950.333,E2 -9950.333} C_VEL
LIN {X 0,Y 561.17,Z 298.745,A -85,B 0,C 180,E1 -9951.342,E2 -9951.342} C_VEL
LIN {X 0,Y 560.711,Z 337.616,A -85,B 0,C 180,E1 -9954.021,E2 -9954.021} C_VEL
LIN {X 0,Y 560.705,Z 347.467,A -85,B 0,C 180,E1 -9954.643,E2 -9954.643} C_VEL
LIN {X 0,Y 558.715,Z 357.173,A -85,B 0,C 180,E1 -9955.006,E2 -9955.006} C_VEL
LIN {X 0,Y 556.167,Z 447.442,A -85,B 0,C 180,E1 -9956.308,E2 -9956.308} C_VEL
LIN {X 0,Y 552.932,Z 527.219,A -85,B 0,C 180,E1 -9957.645,E2 -9957.645} C_VEL
LIN {X 0,Y 548.547,Z 618.27,A -85,B 0,C 180,E1 -9959.383,E2 -9959.383} C_VEL
LIN {X 0,Y 547.462,Z 645.913,A -85,B 0,C 180,E1 -9960.024,E2 -9960.024} C_VEL
LIN {X 0,Y 546.334,Z 667.535,A -85,B 0,C 180,E1 -9960.717,E2 -9960.717} C_VEL
LIN {X 0,Y 544.964,Z 688.15,A -85,B 0,C 180,E1 -9961.567,E2 -9961.567} C_VEL
LIN {X 0,Y 543.313,Z 708.436,A -85,B 0,C 180,E1 -9962.607,E2 -9962.607} C_VEL
LIN {X 0,Y 541.53,Z 727.919,A -85,B 0,C 180,E1 -9963.814,E2 -9963.814} C_VEL
LIN {X 0,Y 539.576,Z 747.236,A -85,B 0,C 180,E1 -9965.241,E2 -9965.241} C_VEL
LIN {X 0,Y 537.609,Z 765.448,A -85,B 0,C 180,E1 -9966.836,E2 -9966.836} C_VEL
LIN {X 0,Y 535.836,Z 781.469,A -85,B 0,C 180,E1 -9968.482,E2 -9968.482} C_VEL
LIN {X 0,Y 534.13,Z 796.811,A -85,B 0,C 180,E1 -9970.325,E2 -9970.325} C_VEL
LIN {X 0,Y 532.617,Z 810.702,A -85,B 0,C 180,E1 -9972.294,E2 -9972.294} C_VEL
LIN {X 0,Y 531.394,Z 822.543,A -85,B 0,C 180,E1 -9974.279,E2 -9974.279} C_VEL
LIN {X 0,Y 530.407,Z 833.084,A -85,B 0,C 180,E1 -9976.37,E2 -9976.37} C_VEL
LIN {X 0,Y 529.678,Z 842.257,A -85,B 0,C 180,E1 -9978.568,E2 -9978.568} C_VEL
LIN {X 0,Y 529.164,Z 849.634,A -85,B 0,C 180,E1 -9980.757,E2 -9980.757} C_VEL
LIN {X 0,Y 528.84,Z 855.487,A -85,B 0,C 180,E1 -9983.042,E2 -9983.042} C_VEL
LIN {X 0,Y 528.68,Z 859.716,A -85,B 0,C 180,E1 -9985.357,E2 -9985.357} C_VEL
LIN {X 0,Y 528.594,Z 862.256,A -85,B 0,C 180,E1 -9987.615,E2 -9987.615} C_VEL
LIN {X 0,Y 528.581,Z 863.187,A -85,B 0,C 180,E1 -9989.892,E2 -9989.892} C_VEL
LIN {X 0,Y 528.591,Z 862.445,A -85,B 0,C 180,E1 -9992.168,E2 -9992.168} C_VEL
LIN {X 0,Y 528.671,Z 859.972,A -85,B 0,C 180,E1 -9994.556,E2 -9994.556} C_VEL
LIN {X 0,Y 528.832,Z 855.965,A -85,B 0,C 180,E1 -9996.841,E2 -9996.841} C_VEL
LIN {X 0,Y 529.123,Z 850.214,A -85,B 0,C 180,E1 -9999.133,E2 -9999.133} C_VEL
LIN {X 0,Y 529.621,Z 842.983,A -85,B 0,C 180,E1 -10001.323,E2 -10001.323} C_VEL
LIN {X 0,Y 530.326,Z 834.004,A -85,B 0,C 180,E1 -10003.52,E2 -10003.52} C_VEL
LIN {X 0,Y 531.287,Z 823.673,A -85,B 0,C 180,E1 -10005.612,E2 -10005.612} C_VEL
LIN {X 0,Y 532.563,Z 811.314,A -85,B 0,C 180,E1 -10007.707,E2 -10007.707} C_VEL
LIN {X 0,Y 534.073,Z 797.357,A -85,B 0,C 180,E1 -10009.694,E2 -10009.694} C_VEL
LIN {X 0,Y 535.744,Z 782.316,A -85,B 0,C 180,E1 -10011.515,E2 -10011.515} C_VEL
LIN {X 0,Y 537.581,Z 765.8,A -85,B 0,C 180,E1 -10013.223,E2 -10013.223} C_VEL
LIN {X 0,Y 539.546,Z 747.653,A -85,B 0,C 180,E1 -10014.819,E2 -10014.819} C_VEL
LIN {X 0,Y 541.418,Z 729.227,A -85,B 0,C 180,E1 -10016.192,E2 -10016.192} C_VEL
LIN {X 0,Y 543.211,Z 710.038,A -85,B 0,C 180,E1 -10017.398,E2 -10017.398} C_VEL
LIN {X 0,Y 544.933,Z 688.869,A -85,B 0,C 180,E1 -10018.494,E2 -10018.494} C_VEL
LIN {X 0,Y 546.395,Z 666.947,A -85,B 0,C 180,E1 -10019.399,E2 -10019.399} C_VEL
LIN {X 0,Y 547.5,Z 645.516,A -85,B 0,C 180,E1 -10020.081,E2 -10020.081} C_VEL
LIN {X 0,Y 548.585,Z 617.9,A -85,B 0,C 180,E1 -10020.719,E2 -10020.719} C_VEL
LIN {X 0,Y 552.911,Z 528.105,A -85,B 0,C 180,E1 -10022.432,E2 -10022.432} C_VEL
LIN {X 0,Y 556.199,Z 447.578,A -85,B 0,C 180,E1 -10023.784,E2 -10023.784} C_VEL
LIN {X 0,Y 558.848,Z 355.951,A -85,B 0,C 180,E1 -10025.116,E2 -10025.116} C_VEL
LIN {X 0,Y 560.858,Z 347.053,A -85,B 0,C 180,E1 -10025.471,E2 -10025.471} C_VEL
LIN {X 0,Y 560.927,Z 311.586,A -85,B 0,C 180,E1 -10027.844,E2 -10027.844} C_VEL
LIN {X 0,Y 561.314,Z 290.462,A -85,B 0,C 180,E1 -10029.366,E2 -10029.366} C_VEL
LIN {X 0,Y 552.958,Z 268.273,A -85,B 0,C 180,E1 -10031.84,E2 -10031.84} C_VEL
LIN {X 0,Y 544.509,Z 248.807,A -85,B 0,C 180,E1 -10034.11,E2 -10034.11} C_VEL
LIN {X 0,Y 536.433,Z 232.49,A -85,B 0,C 180,E1 -10036.1,E2 -10036.1} C_VEL
LIN {X 0,Y 531.595,Z 223.54,A -85,B 0,C 180,E1 -10037.233,E2 -10037.233} C_VEL
LIN {X 0,Y 529.865,Z 220.226,A -85,B 0,C 180,E1 -10037.648,E2 -10037.648} C_VEL
LIN {X 0,Y 529.686,Z 219.255,A -85,B 0,C 180,E1 -10037.756,E2 -10037.756} C_VEL
LIN {X 0,Y 529.667,Z 219.256,A -85,B 0,C 180,E1 -10041.19,E2 -10041.19} C_VEL
LIN {X 0,Y 529.684,Z 219.25,A -85,B 0,C 180,E1 -10044.636,E2 -10044.636} C_VEL
LIN {X 0,Y 529.678,Z 219.237,A -85,B 0,C 180,E1 -10048.091,E2 -10048.091} C_VEL
LIN {X 0,Y 529.675,Z 219.226,A -85,B 0,C 180,E1 -10051.471,E2 -10051.471} C_VEL
LIN {X 0,Y 529.676,Z 219.243,A -85,B 0,C 180,E1 -10054.985,E2 -10054.985} C_VEL
LIN {X 0,Y 529.677,Z 219.248,A -85,B 0,C 180,E1 -10058.401,E2 -10058.401} C_VEL
LIN {X 0,Y 529.679,Z 219.217,A -85,B 0,C 180,E1 -10061.852,E2 -10061.852} C_VEL
LIN {X 0,Y 529.678,Z 219.248,A -85,B 0,C 180,E1 -10065.236,E2 -10065.236} C_VEL
LIN {X 0,Y 529.673,Z 219.224,A -85,B 0,C 180,E1 -10068.678,E2 -10068.678} C_VEL
LIN {X 0,Y 529.669,Z 219.239,A -85,B 0,C 180,E1 -10072.188,E2 -10072.188} C_VEL
LIN {X 0,Y 529.678,Z 219.231,A -85,B 0,C 180,E1 -10075.561,E2 -10075.561} C_VEL
LIN {X 0,Y 529.686,Z 219.234,A -85,B 0,C 180,E1 -10079.027,E2 -10079.027} C_VEL
LIN {X 0,Y 529.66,Z 219.243,A -85,B 0,C 180,E1 -10082.489,E2 -10082.489} C_VEL
LIN {X 0,Y 529.674,Z 219.223,A -85,B 0,C 180,E1 -10085.96,E2 -10085.96} C_VEL
LIN {X 0,Y 529.685,Z 219.242,A -85,B 0,C 180,E1 -10089.453,E2 -10089.453} C_VEL
LIN {X 0,Y 529.667,Z 219.249,A -85,B 0,C 180,E1 -10092.871,E2 -10092.871} C_VEL
LIN {X 0,Y 529.655,Z 219.254,A -85,B 0,C 180,E1 -10096.337,E2 -10096.337} C_VEL
LIN {X 0,Y 529.687,Z 219.251,A -85,B 0,C 180,E1 -10099.749,E2 -10099.749} C_VEL
LIN {X 0,Y 529.678,Z 219.252,A -85,B 0,C 180,E1 -10103.172,E2 -10103.172} C_VEL
LIN {X 0,Y 529.649,Z 219.246,A -85,B 0,C 180,E1 -10106.578,E2 -10106.578} C_VEL
LIN {X 0,Y 529.683,Z 219.247,A -85,B 0,C 180,E1 -10109.95,E2 -10109.95} C_VEL
LIN {X 0,Y 529.677,Z 219.248,A -85,B 0,C 180,E1 -10113.321,E2 -10113.321} C_VEL
LIN {X 0,Y 529.66,Z 219.289,A -85,B 0,C 180,E1 -10114.266,E2 -10114.266} C_VEL
LIN {X 0,Y 530.757,Z 222.44,A -85,B 0,C 180,E1 -10114.676,E2 -10114.676} C_VEL
LIN {X 0,Y 532.266,Z 225.006,A -85,B 0,C 180,E1 -10115.088,E2 -10115.088} C_VEL
LIN {X 0,Y 540.989,Z 242.005,A -85,B 0,C 180,E1 -10117.542,E2 -10117.542} C_VEL
LIN {X 0,Y 551.488,Z 262.944,A -85,B 0,C 180,E1 -10120.336,E2 -10120.336} C_VEL
LIN {X 0,Y 563.478,Z 287.574,A -85,B 0,C 180,E1 -10123.319,E2 -10123.319} C_VEL
LIN {X 0,Y 567.952,Z 297.375,A -85,B 0,C 180,E1 -10124.412,E2 -10124.412} C_VEL
LIN {X 0,Y 566.382,Z 313.036,A -85,B 0,C 180,E1 -10125.322,E2 -10125.322} C_VEL
LIN {X 0,Y 569.212,Z 339.156,A -85,B 0,C 180,E1 -10126.019,E2 -10126.019} C_VEL
LIN {X 0,Y 561.49,Z 578.773,A -85,B 0,C 180,E1 -10129.621,E2 -10129.621} C_VEL
LIN {X 0,Y 558.297,Z 692.879,A -85,B 0,C 180,E1 -10131.299,E2 -10131.299} C_VEL
LIN {X 0,Y 556.902,Z 717.524,A -85,B 0,C 180,E1 -10131.836,E2 -10131.836} C_VEL
LIN {X 0,Y 555.258,Z 740.84,A -85,B 0,C 180,E1 -10132.507,E2 -10132.507} C_VEL
LIN {X 0,Y 553.211,Z 764.053,A -85,B 0,C 180,E1 -10133.37,E2 -10133.37} C_VEL
LIN {X 0,Y 550.987,Z 786.469,A -85,B 0,C 180,E1 -10134.372,E2 -10134.372} C_VEL
LIN {X 0,Y 548.466,Z 808.771,A -85,B 0,C 180,E1 -10135.587,E2 -10135.587} C_VEL
LIN {X 0,Y 545.954,Z 829.862,A -85,B 0,C 180,E1 -10136.922,E2 -10136.922} C_VEL
LIN {X 0,Y 543.365,Z 850.07,A -85,B 0,C 180,E1 -10138.431,E2 -10138.431} C_VEL
LIN {X 0,Y 540.876,Z 869.234,A -85,B 0,C 180,E1 -10140.057,E2 -10140.057} C_VEL
LIN {X 0,Y 538.406,Z 887.394,A -85,B 0,C 180,E1 -10141.855,E2 -10141.855} C_VEL
LIN {X 0,Y 536.191,Z 904.525,A -85,B 0,C 180,E1 -10143.771,E2 -10143.771} C_VEL
LIN {X 0,Y 534.175,Z 920.177,A -85,B 0,C 180,E1 -10145.799,E2 -10145.799} C_VEL
LIN {X 0,Y 532.465,Z 934.734,A -85,B 0,C 180,E1 -10147.94,E2 -10147.94} C_VEL
LIN {X 0,Y 531.024,Z 947.861,A -85,B 0,C 180,E1 -10150.188,E2 -10150.188} C_VEL
LIN {X 0,Y 529.956,Z 959.277,A -85,B 0,C 180,E1 -10152.43,E2 -10152.43} C_VEL
LIN {X 0,Y 529.085,Z 970.28,A -85,B 0,C 180,E1 -10154.995,E2 -10154.995} C_VEL
LIN {X 0,Y 528.596,Z 978.281,A -85,B 0,C 180,E1 -10157.214,E2 -10157.214} C_VEL
LIN {X 0,Y 528.245,Z 986.314,A -85,B 0,C 180,E1 -10159.971,E2 -10159.971} C_VEL
LIN {X 0,Y 528.098,Z 991.25,A -85,B 0,C 180,E1 -10162.165,E2 -10162.165} C_VEL
LIN {X 0,Y 528.05,Z 995.309,A -85,B 0,C 180,E1 -10164.567,E2 -10164.567} C_VEL
LIN {X 0,Y 528.058,Z 997.854,A -85,B 0,C 180,E1 -10167.07,E2 -10167.07} C_VEL
